LIN {X 0,Y 496.76,Z 265.856,A -85,B 0,C 180,E1 24154.304,E2 24154.304} C_VEL
LIN {X 0,Y 496.744,Z 265.83,A -85,B 0,C 180,E1 24150.745,E2 24150.745} C_VEL
LIN {X 0,Y 496.768,Z 265.857,A -85,B 0,C 180,E1 24147.316,E2 24147.316} C_VEL
LIN {X 0,Y 496.772,Z 265.855,A -85,B 0,C 180,E1 24143.686,E2 24143.686} C_VEL
LIN {X 0,Y 496.741,Z 265.856,A -85,B 0,C 180,E1 24140.256,E2 24140.256} C_VEL
LIN {X 0,Y 496.732,Z 265.859,A -85,B 0,C 180,E1 24136.645,E2 24136.645} C_VEL
LIN {X 0,Y 496.759,Z 265.856,A -85,B 0,C 180,E1 24133.147,E2 24133.147} C_VEL
LIN {X 0,Y 496.765,Z 265.845,A -85,B 0,C 180,E1 24129.617,E2 24129.617} C_VEL
LIN {X 0,Y 496.72,Z 265.85,A -85,B 0,C 180,E1 24126.24,E2 24126.24} C_VEL
LIN {X 0,Y 496.719,Z 265.855,A -85,B 0,C 180,E1 24122.654,E2 24122.654} C_VEL
LIN {X 0,Y 496.76,Z 265.86,A -85,B 0,C 180,E1 24119.193,E2 24119.193} C_VEL
LIN {X 0,Y 496.733,Z 265.855,A -85,B 0,C 180,E1 24115.729,E2 24115.729} C_VEL
LIN {X 0,Y 496.699,Z 265.854,A -85,B 0,C 180,E1 24112.365,E2 24112.365} C_VEL
LIN {X 0,Y 496.73,Z 265.851,A -85,B 0,C 180,E1 24108.976,E2 24108.976} C_VEL
LIN {X 0,Y 496.727,Z 265.86,A -85,B 0,C 180,E1 24105.546,E2 24105.546} C_VEL
LIN {X 0,Y 496.69,Z 265.861,A -85,B 0,C 180,E1 24102.183,E2 24102.183} C_VEL
LIN {X 0,Y 496.72,Z 265.86,A -85,B 0,C 180,E1 24098.742,E2 24098.742} C_VEL
LIN {X 0,Y 496.747,Z 265.859,A -85,B 0,C 180,E1 24095.377,E2 24095.377} C_VEL
LIN {X 0,Y 496.706,Z 265.861,A -85,B 0,C 180,E1 24092.029,E2 24092.029} C_VEL
LIN {X 0,Y 496.724,Z 265.83,A -85,B 0,C 180,E1 24088.578,E2 24088.578} C_VEL
LIN {X 0,Y 496.766,Z 265.852,A -85,B 0,C 180,E1 24085.137,E2 24085.137} C_VEL
LIN {X 0,Y 496.729,Z 265.852,A -85,B 0,C 180,E1 24081.686,E2 24081.686} C_VEL
LIN {X 0,Y 496.723,Z 265.835,A -85,B 0,C 180,E1 24078.138,E2 24078.138} C_VEL
LIN {X 0,Y 496.761,Z 265.831,A -85,B 0,C 180,E1 24074.724,E2 24074.724} C_VEL
LIN {X 0,Y 496.765,Z 266.073,A -85,B 0,C 180,E1 24073.733,E2 24073.733} C_VEL
LIN {X 0,Y 498.202,Z 269.541,A -85,B 0,C 180,E1 24073.238,E2 24073.238} C_VEL
LIN {X 0,Y 506.88,Z 288.7,A -85,B 0,C 180,E1 24070.845,E2 24070.845} C_VEL
LIN {X 0,Y 512.314,Z 301.504,A -85,B 0,C 180,E1 24069.366,E2 24069.366} C_VEL
LIN {X 0,Y 512.445,Z 304.432,A -85,B 0,C 180,E1 24069.211,E2 24069.211} C_VEL
LIN {X 0,Y 515.554,Z 323.753,A -85,B 0,C 180,E1 24068.621,E2 24068.621} C_VEL
LIN {X 0,Y 512.644,Z 536.307,A -85,B 0,C 180,E1 24065.312,E2 24065.312} C_VEL
LIN {X 0,Y 511.651,Z 609.629,A -85,B 0,C 180,E1 24064.168,E2 24064.168} C_VEL
LIN {X 0,Y 510.839,Z 630.079,A -85,B 0,C 180,E1 24063.658,E2 24063.658} C_VEL
LIN {X 0,Y 509.734,Z 651.77,A -85,B 0,C 180,E1 24062.909,E2 24062.909} C_VEL
LIN {X 0,Y 508.491,Z 672.18,A -85,B 0,C 180,E1 24061.999,E2 24061.999} C_VEL
LIN {X 0,Y 507.033,Z 691.752,A -85,B 0,C 180,E1 24060.91,E2 24060.91} C_VEL
LIN {X 0,Y 505.464,Z 711.909,A -85,B 0,C 180,E1 24059.555,E2 24059.555} C_VEL
LIN {X 0,Y 503.931,Z 730.052,A -85,B 0,C 180,E1 24058.113,E2 24058.113} C_VEL
LIN {X 0,Y 502.359,Z 748.13,A -85,B 0,C 180,E1 24056.409,E2 24056.409} C_VEL
LIN {X 0,Y 500.871,Z 765.167,A -85,B 0,C 180,E1 24054.532,E2 24054.532} C_VEL
LIN {X 0,Y 499.613,Z 780.33,A -85,B 0,C 180,E1 24052.596,E2 24052.596} C_VEL
LIN {X 0,Y 498.485,Z 794.868,A -85,B 0,C 180,E1 24050.426,E2 24050.426} C_VEL
LIN {X 0,Y 497.624,Z 807.187,A -85,B 0,C 180,E1 24048.266,E2 24048.266} C_VEL
LIN {X 0,Y 496.93,Z 818.784,A -85,B 0,C 180,E1 24045.881,E2 24045.881} C_VEL
LIN {X 0,Y 496.465,Z 828.431,A -85,B 0,C 180,E1 24043.51,E2 24043.51} C_VEL
LIN {X 0,Y 496.159,Z 836.434,A -85,B 0,C 180,E1 24041.069,E2 24041.069} C_VEL
LIN {X 0,Y 495.997,Z 842.892,A -85,B 0,C 180,E1 24038.579,E2 24038.579} C_VEL
LIN {X 0,Y 495.935,Z 847.43,A -85,B 0,C 180,E1 24036.25,E2 24036.25} C_VEL
LIN {X 0,Y 495.907,Z 850.56,A -85,B 0,C 180,E1 24033.815,E2 24033.815} C_VEL
LIN {X 0,Y 495.902,Z 852.237,A -85,B 0,C 180,E1 24031.386,E2 24031.386} C_VEL
LIN {X 0,Y 495.909,Z 852.327,A -85,B 0,C 180,E1 24029.076,E2 24029.076} C_VEL
LIN {X 0,Y 495.911,Z 850.898,A -85,B 0,C 180,E1 24026.532,E2 24026.532} C_VEL
LIN {X 0,Y 495.931,Z 847.98,A -85,B 0,C 180,E1 24024.098,E2 24024.098} C_VEL
LIN {X 0,Y 496,Z 843.399,A -85,B 0,C 180,E1 24021.655,E2 24021.655} C_VEL
LIN {X 0,Y 496.141,Z 837.235,A -85,B 0,C 180,E1 24019.198,E2 24019.198} C_VEL
LIN {X 0,Y 496.403,Z 829.665,A -85,B 0,C 180,E1 24016.844,E2 24016.844} C_VEL
LIN {X 0,Y 496.836,Z 820.328,A -85,B 0,C 180,E1 24014.476,E2 24014.476} C_VEL
LIN {X 0,Y 497.459,Z 809.727,A -85,B 0,C 180,E1 24012.212,E2 24012.212} C_VEL
LIN {X 0,Y 498.274,Z 797.763,A -85,B 0,C 180,E1 24010.055,E2 24010.055} C_VEL
LIN {X 0,Y 499.339,Z 783.717,A -85,B 0,C 180,E1 24007.887,E2 24007.887} C_VEL
LIN {X 0,Y 500.624,Z 768.208,A -85,B 0,C 180,E1 24005.832,E2 24005.832} C_VEL
LIN {X 0,Y 501.995,Z 752.25,A -85,B 0,C 180,E1 24004.012,E2 24004.012} C_VEL
LIN {X 0,Y 503.516,Z 734.772,A -85,B 0,C 180,E1 24002.312,E2 24002.312} C_VEL
LIN {X 0,Y 505.136,Z 715.755,A -85,B 0,C 180,E1 24000.732,E2 24000.732} C_VEL
LIN {X 0,Y 506.688,Z 696.76,A -85,B 0,C 180,E1 23999.396,E2 23999.396} C_VEL
LIN {X 0,Y 508.188,Z 676.137,A -85,B 0,C 180,E1 23998.207,E2 23998.207} C_VEL
LIN {X 0,Y 509.534,Z 655.455,A -85,B 0,C 180,E1 23997.242,E2 23997.242} C_VEL
LIN {X 0,Y 510.643,Z 634.593,A -85,B 0,C 180,E1 23996.473,E2 23996.473} C_VEL
LIN {X 0,Y 511.474,Z 614.158,A -85,B 0,C 180,E1 23995.932,E2 23995.932} C_VEL
LIN {X 0,Y 512.059,Z 584.884,A -85,B 0,C 180,E1 23995.426,E2 23995.426} C_VEL
LIN {X 0,Y 514.855,Z 371.498,A -85,B 0,C 180,E1 23992.134,E2 23992.134} C_VEL
LIN {X 0,Y 515.386,Z 321.569,A -85,B 0,C 180,E1 23991.328,E2 23991.328} C_VEL
LIN {X 0,Y 512.272,Z 302.49,A -85,B 0,C 180,E1 23990.703,E2 23990.703} C_VEL
LIN {X 0,Y 512.096,Z 300.679,A -85,B 0,C 180,E1 23990.552,E2 23990.552} C_VEL
LIN {X 0,Y 502.008,Z 277.659,A -85,B 0,C 180,E1 23987.809,E2 23987.809} C_VEL
LIN {X 0,Y 496.796,Z 266.243,A -85,B 0,C 180,E1 23986.311,E2 23986.311} C_VEL
LIN {X 0,Y 496.743,Z 265.832,A -85,B 0,C 180,E1 23985.537,E2 23985.537} C_VEL
LIN {X 0,Y 496.723,Z 265.836,A -85,B 0,C 180,E1 23982.034,E2 23982.034} C_VEL
LIN {X 0,Y 496.753,Z 265.852,A -85,B 0,C 180,E1 23978.606,E2 23978.606} C_VEL
LIN {X 0,Y 496.758,Z 265.848,A -85,B 0,C 180,E1 23975.145,E2 23975.145} C_VEL
LIN {X 0,Y 496.712,Z 265.833,A -85,B 0,C 180,E1 23971.694,E2 23971.694} C_VEL
LIN {X 0,Y 496.713,Z 265.861,A -85,B 0,C 180,E1 23968.101,E2 23968.101} C_VEL
LIN {X 0,Y 496.76,Z 265.86,A -85,B 0,C 180,E1 23964.749,E2 23964.749} C_VEL
LIN {X 0,Y 496.712,Z 265.86,A -85,B 0,C 180,E1 23961.367,E2 23961.367} C_VEL
LIN {X 0,Y 496.695,Z 265.861,A -85,B 0,C 180,E1 23957.938,E2 23957.938} C_VEL
LIN {X 0,Y 496.733,Z 265.858,A -85,B 0,C 180,E1 23954.496,E2 23954.496} C_VEL
LIN {X 0,Y 496.725,Z 265.851,A -85,B 0,C 180,E1 23951.024,E2 23951.024} C_VEL
LIN {X 0,Y 496.695,Z 265.855,A -85,B 0,C 180,E1 23947.635,E2 23947.635} C_VEL
LIN {X 0,Y 496.721,Z 265.856,A -85,B 0,C 180,E1 23944.155,E2 23944.155} C_VEL
LIN {X 0,Y 496.767,Z 265.859,A -85,B 0,C 180,E1 23940.692,E2 23940.692} C_VEL
LIN {X 0,Y 496.72,Z 265.855,A -85,B 0,C 180,E1 23937.231,E2 23937.231} C_VEL
LIN {X 0,Y 496.717,Z 265.85,A -85,B 0,C 180,E1 23933.759,E2 23933.759} C_VEL
LIN {X 0,Y 496.764,Z 265.846,A -85,B 0,C 180,E1 23930.383,E2 23930.383} C_VEL
LIN {X 0,Y 496.753,Z 265.858,A -85,B 0,C 180,E1 23926.853,E2 23926.853} C_VEL
LIN {X 0,Y 496.728,Z 265.858,A -85,B 0,C 180,E1 23923.391,E2 23923.391} C_VEL
LIN {X 0,Y 496.745,Z 265.855,A -85,B 0,C 180,E1 23919.867,E2 23919.867} C_VEL
LIN {X 0,Y 496.771,Z 265.856,A -85,B 0,C 180,E1 23916.388,E2 23916.388} C_VEL
LIN {X 0,Y 496.761,Z 265.853,A -85,B 0,C 180,E1 23912.813,E2 23912.813} C_VEL
LIN {X 0,Y 496.74,Z 265.832,A -85,B 0,C 180,E1 23909.386,E2 23909.386} C_VEL
LIN {X 0,Y 496.762,Z 265.855,A -85,B 0,C 180,E1 23905.814,E2 23905.814} C_VEL
LIN {X 0,Y 496.762,Z 265.83,A -85,B 0,C 180,E1 23902.274,E2 23902.274} C_VEL
LIN {X 0,Y 496.768,Z 265.836,A -85,B 0,C 180,E1 23898.687,E2 23898.687} C_VEL
LIN {X 0,Y 496.758,Z 265.857,A -85,B 0,C 180,E1 23895.05,E2 23895.05} C_VEL
LIN {X 0,Y 496.765,Z 265.859,A -85,B 0,C 180,E1 23891.466,E2 23891.466} C_VEL
LIN {X 0,Y 496.819,Z 266.17,A -85,B 0,C 180,E1 23890.648,E2 23890.648} C_VEL
LIN {X 0,Y 505.817,Z 287.439,A -85,B 0,C 180,E1 23887.75,E2 23887.75} C_VEL
LIN {X 0,Y 507.172,Z 290.873,A -85,B 0,C 180,E1 23887.316,E2 23887.316} C_VEL
LIN {X 0,Y 507.772,Z 294.918,A -85,B 0,C 180,E1 23886.901,E2 23886.901} C_VEL
LIN {X 0,Y 506.892,Z 301.33,A -85,B 0,C 180,E1 23886.41,E2 23886.41} C_VEL
LIN {X 0,Y 502.273,Z 317.887,A -85,B 0,C 180,E1 23885.352,E2 23885.352} C_VEL
LIN {X 0,Y 501.917,Z 320.739,A -85,B 0,C 180,E1 23885.132,E2 23885.132} C_VEL
LIN {X 0,Y 501.604,Z 327.881,A -85,B 0,C 180,E1 23884.576,E2 23884.576} C_VEL
LIN {X 0,Y 505.479,Z 350.471,A -85,B 0,C 180,E1 23883.865,E2 23883.865} C_VEL
LIN {X 0,Y 502.237,Z 583.059,A -85,B 0,C 180,E1 23880.294,E2 23880.294} C_VEL
LIN {X 0,Y 501.63,Z 603.88,A -85,B 0,C 180,E1 23879.854,E2 23879.854} C_VEL
LIN {X 0,Y 500.665,Z 623.703,A -85,B 0,C 180,E1 23879.22,E2 23879.22} C_VEL
LIN {X 0,Y 499.463,Z 643.041,A -85,B 0,C 180,E1 23878.387,E2 23878.387} C_VEL
LIN {X 0,Y 498.088,Z 661.685,A -85,B 0,C 180,E1 23877.366,E2 23877.366} C_VEL
LIN {X 0,Y 496.606,Z 679.561,A -85,B 0,C 180,E1 23876.163,E2 23876.163} C_VEL
LIN {X 0,Y 495.015,Z 697.298,A -85,B 0,C 180,E1 23874.715,E2 23874.715} C_VEL
LIN {X 0,Y 493.413,Z 714.532,A -85,B 0,C 180,E1 23873.022,E2 23873.022} C_VEL
LIN {X 0,Y 491.984,Z 730.027,A -85,B 0,C 180,E1 23871.207,E2 23871.207} C_VEL
LIN {X 0,Y 490.748,Z 744.004,A -85,B 0,C 180,E1 23869.272,E2 23869.272} C_VEL
LIN {X 0,Y 489.675,Z 758.025,A -85,B 0,C 180,E1 23866.977,E2 23866.977} C_VEL
LIN {X 0,Y 488.978,Z 769.274,A -85,B 0,C 180,E1 23864.809,E2 23864.809} C_VEL
LIN {X 0,Y 488.472,Z 779.247,A -85,B 0,C 180,E1 23862.478,E2 23862.478} C_VEL
LIN {X 0,Y 488.166,Z 787.28,A -85,B 0,C 180,E1 23860.145,E2 23860.145} C_VEL
LIN {X 0,Y 488.015,Z 793.376,A -85,B 0,C 180,E1 23857.89,E2 23857.89} C_VEL
LIN {X 0,Y 487.931,Z 798.008,A -85,B 0,C 180,E1 23855.527,E2 23855.527} C_VEL
LIN {X 0,Y 487.909,Z 800.962,A -85,B 0,C 180,E1 23853.172,E2 23853.172} C_VEL
LIN {X 0,Y 487.907,Z 802.359,A -85,B 0,C 180,E1 23850.704,E2 23850.704} C_VEL
LIN {X 0,Y 487.902,Z 802.102,A -85,B 0,C 180,E1 23848.356,E2 23848.356} C_VEL
LIN {X 0,Y 487.918,Z 800.255,A -85,B 0,C 180,E1 23846.005,E2 23846.005} C_VEL
LIN {X 0,Y 487.953,Z 796.675,A -85,B 0,C 180,E1 23843.622,E2 23843.622} C_VEL
LIN {X 0,Y 488.053,Z 791.516,A -85,B 0,C 180,E1 23841.281,E2 23841.281} C_VEL
LIN {X 0,Y 488.258,Z 784.528,A -85,B 0,C 180,E1 23838.902,E2 23838.902} C_VEL
LIN {X 0,Y 488.621,Z 776.086,A -85,B 0,C 180,E1 23836.631,E2 23836.631} C_VEL
LIN {X 0,Y 489.198,Z 765.655,A -85,B 0,C 180,E1 23834.349,E2 23834.349} C_VEL
LIN {X 0,Y 490.041,Z 752.956,A -85,B 0,C 180,E1 23832.056,E2 23832.056} C_VEL
LIN {X 0,Y 491.123,Z 739.689,A -85,B 0,C 180,E1 23830,E2 23830} C_VEL
LIN {X 0,Y 492.441,Z 724.859,A -85,B 0,C 180,E1 23828.063,E2 23828.063} C_VEL
LIN {X 0,Y 493.859,Z 709.496,A -85,B 0,C 180,E1 23826.368,E2 23826.368} C_VEL
LIN {X 0,Y 495.425,Z 692.653,A -85,B 0,C 180,E1 23824.797,E2 23824.797} C_VEL
LIN {X 0,Y 497,Z 674.858,A -85,B 0,C 180,E1 23823.41,E2 23823.41} C_VEL
LIN {X 0,Y 498.465,Z 657.122,A -85,B 0,C 180,E1 23822.267,E2 23822.267} C_VEL
LIN {X 0,Y 499.773,Z 638.535,A -85,B 0,C 180,E1 23821.306,E2 23821.306} C_VEL
LIN {X 0,Y 500.896,Z 619.188,A -85,B 0,C 180,E1 23820.53,E2 23820.53} C_VEL
LIN {X 0,Y 501.8,Z 598.35,A -85,B 0,C 180,E1 23819.922,E2 23819.922} C_VEL
LIN {X 0,Y 502.38,Z 574.514,A -85,B 0,C 180,E1 23819.48,E2 23819.48} C_VEL
LIN {X 0,Y 505.455,Z 349.374,A -85,B 0,C 180,E1 23816.024,E2 23816.024} C_VEL
LIN {X 0,Y 501.532,Z 326.8,A -85,B 0,C 180,E1 23815.274,E2 23815.274} C_VEL
LIN {X 0,Y 503.113,Z 301.394,A -85,B 0,C 180,E1 23813.169,E2 23813.169} C_VEL
LIN {X 0,Y 495.083,Z 281.538,A -85,B 0,C 180,E1 23810.578,E2 23810.578} C_VEL
LIN {X 0,Y 488.87,Z 267.138,A -85,B 0,C 180,E1 23808.498,E2 23808.498} C_VEL
LIN {X 0,Y 488.825,Z 266.818,A -85,B 0,C 180,E1 23806.426,E2 23806.426} C_VEL
LIN {X 0,Y 488.818,Z 266.819,A -85,B 0,C 180,E1 23802.924,E2 23802.924} C_VEL
LIN {X 0,Y 488.831,Z 266.843,A -85,B 0,C 180,E1 23799.352,E2 23799.352} C_VEL
LIN {X 0,Y 488.824,Z 266.832,A -85,B 0,C 180,E1 23795.659,E2 23795.659} C_VEL
LIN {X 0,Y 488.823,Z 266.82,A -85,B 0,C 180,E1 23792.128,E2 23792.128} C_VEL
LIN {X 0,Y 488.807,Z 266.847,A -85,B 0,C 180,E1 23788.597,E2 23788.597} C_VEL
LIN {X 0,Y 488.817,Z 266.846,A -85,B 0,C 180,E1 23785.026,E2 23785.026} C_VEL
LIN {X 0,Y 488.832,Z 266.838,A -85,B 0,C 180,E1 23781.467,E2 23781.467} C_VEL
LIN {X 0,Y 488.822,Z 266.836,A -85,B 0,C 180,E1 23777.868,E2 23777.868} C_VEL
LIN {X 0,Y 488.792,Z 266.837,A -85,B 0,C 180,E1 23774.331,E2 23774.331} C_VEL
LIN {X 0,Y 488.79,Z 266.836,A -85,B 0,C 180,E1 23770.728,E2 23770.728} C_VEL
LIN {X 0,Y 488.828,Z 266.842,A -85,B 0,C 180,E1 23767.252,E2 23767.252} C_VEL
LIN {X 0,Y 488.807,Z 266.846,A -85,B 0,C 180,E1 23763.753,E2 23763.753} C_VEL
LIN {X 0,Y 488.771,Z 266.847,A -85,B 0,C 180,E1 23760.352,E2 23760.352} C_VEL
LIN {X 0,Y 488.785,Z 266.842,A -85,B 0,C 180,E1 23756.834,E2 23756.834} C_VEL
LIN {X 0,Y 488.827,Z 266.838,A -85,B 0,C 180,E1 23753.305,E2 23753.305} C_VEL
LIN {X 0,Y 488.77,Z 266.85,A -85,B 0,C 180,E1 23749.868,E2 23749.868} C_VEL
LIN {X 0,Y 488.752,Z 266.85,A -85,B 0,C 180,E1 23746.336,E2 23746.336} C_VEL
LIN {X 0,Y 488.794,Z 266.85,A -85,B 0,C 180,E1 23742.992,E2 23742.992} C_VEL
LIN {X 0,Y 488.79,Z 266.844,A -85,B 0,C 180,E1 23739.526,E2 23739.526} C_VEL
LIN {X 0,Y 488.762,Z 266.847,A -85,B 0,C 180,E1 23736.106,E2 23736.106} C_VEL
LIN {X 0,Y 488.783,Z 266.849,A -85,B 0,C 180,E1 23732.594,E2 23732.594} C_VEL
LIN {X 0,Y 488.831,Z 266.813,A -85,B 0,C 180,E1 23729.11,E2 23729.11} C_VEL
LIN {X 0,Y 488.801,Z 266.851,A -85,B 0,C 180,E1 23725.52,E2 23725.52} C_VEL
LIN {X 0,Y 488.779,Z 266.834,A -85,B 0,C 180,E1 23721.995,E2 23721.995} C_VEL
LIN {X 0,Y 488.799,Z 266.819,A -85,B 0,C 180,E1 23718.473,E2 23718.473} C_VEL
LIN {X 0,Y 488.829,Z 266.819,A -85,B 0,C 180,E1 23714.951,E2 23714.951} C_VEL
LIN {X 0,Y 488.877,Z 267.302,A -85,B 0,C 180,E1 23714.435,E2 23714.435} C_VEL
LIN {X 0,Y 497.975,Z 287.252,A -85,B 0,C 180,E1 23711.804,E2 23711.804} C_VEL
LIN {X 0,Y 505.312,Z 303.93,A -85,B 0,C 180,E1 23709.827,E2 23709.827} C_VEL
LIN {X 0,Y 506.077,Z 306.304,A -85,B 0,C 180,E1 23709.716,E2 23709.716} C_VEL
LIN {X 0,Y 509.065,Z 325.262,A -85,B 0,C 180,E1 23709.128,E2 23709.128} C_VEL
LIN {X 0,Y 505.837,Z 535.278,A -85,B 0,C 180,E1 23705.801,E2 23705.801} C_VEL
LIN {X 0,Y 504.715,Z 609.546,A -85,B 0,C 180,E1 23704.623,E2 23704.623} C_VEL
LIN {X 0,Y 503.838,Z 631.178,A -85,B 0,C 180,E1 23704.08,E2 23704.08} C_VEL
LIN {X 0,Y 502.733,Z 652.958,A -85,B 0,C 180,E1 23703.327,E2 23703.327} C_VEL
LIN {X 0,Y 501.529,Z 673.25,A -85,B 0,C 180,E1 23702.43,E2 23702.43} C_VEL
LIN {X 0,Y 500.052,Z 691.983,A -85,B 0,C 180,E1 23701.374,E2 23701.374} C_VEL
LIN {X 0,Y 498.309,Z 712.502,A -85,B 0,C 180,E1 23699.974,E2 23699.974} C_VEL
LIN {X 0,Y 496.645,Z 730.759,A -85,B 0,C 180,E1 23698.498,E2 23698.498} C_VEL
LIN {X 0,Y 494.933,Z 748.869,A -85,B 0,C 180,E1 23696.758,E2 23696.758} C_VEL
LIN {X 0,Y 493.328,Z 765.673,A -85,B 0,C 180,E1 23694.869,E2 23694.869} C_VEL
LIN {X 0,Y 491.921,Z 781.18,A -85,B 0,C 180,E1 23692.843,E2 23692.843} C_VEL
LIN {X 0,Y 490.705,Z 795.633,A -85,B 0,C 180,E1 23690.64,E2 23690.64} C_VEL
LIN {X 0,Y 489.724,Z 808.455,A -85,B 0,C 180,E1 23688.325,E2 23688.325} C_VEL
LIN {X 0,Y 488.981,Z 819.813,A -85,B 0,C 180,E1 23685.902,E2 23685.902} C_VEL
LIN {X 0,Y 488.486,Z 829.26,A -85,B 0,C 180,E1 23683.493,E2 23683.493} C_VEL
LIN {X 0,Y 488.176,Z 836.882,A -85,B 0,C 180,E1 23681.1,E2 23681.1} C_VEL
LIN {X 0,Y 488.003,Z 843.146,A -85,B 0,C 180,E1 23678.602,E2 23678.602} C_VEL
LIN {X 0,Y 487.937,Z 847.823,A -85,B 0,C 180,E1 23676.117,E2 23676.117} C_VEL
LIN {X 0,Y 487.908,Z 850.799,A -85,B 0,C 180,E1 23673.63,E2 23673.63} C_VEL
LIN {X 0,Y 487.911,Z 852.304,A -85,B 0,C 180,E1 23671.057,E2 23671.057} C_VEL
LIN {X 0,Y 487.905,Z 852.258,A -85,B 0,C 180,E1 23668.708,E2 23668.708} C_VEL
LIN {X 0,Y 487.907,Z 850.671,A -85,B 0,C 180,E1 23666.24,E2 23666.24} C_VEL
LIN {X 0,Y 487.937,Z 847.633,A -85,B 0,C 180,E1 23663.765,E2 23663.765} C_VEL
LIN {X 0,Y 488.003,Z 843.145,A -85,B 0,C 180,E1 23661.398,E2 23661.398} C_VEL
LIN {X 0,Y 488.184,Z 836.663,A -85,B 0,C 180,E1 23658.826,E2 23658.826} C_VEL
LIN {X 0,Y 488.51,Z 828.85,A -85,B 0,C 180,E1 23656.387,E2 23656.387} C_VEL
LIN {X 0,Y 489.028,Z 819.118,A -85,B 0,C 180,E1 23653.935,E2 23653.935} C_VEL
LIN {X 0,Y 489.77,Z 807.821,A -85,B 0,C 180,E1 23651.553,E2 23651.553} C_VEL
LIN {X 0,Y 490.704,Z 795.633,A -85,B 0,C 180,E1 23649.36,E2 23649.36} C_VEL
LIN {X 0,Y 491.921,Z 781.18,A -85,B 0,C 180,E1 23647.157,E2 23647.157} C_VEL
LIN {X 0,Y 493.328,Z 765.674,A -85,B 0,C 180,E1 23645.131,E2 23645.131} C_VEL
LIN {X 0,Y 494.947,Z 748.704,A -85,B 0,C 180,E1 23643.226,E2 23643.226} C_VEL
LIN {X 0,Y 496.644,Z 730.761,A -85,B 0,C 180,E1 23641.502,E2 23641.502} C_VEL
LIN {X 0,Y 498.311,Z 712.507,A -85,B 0,C 180,E1 23640.026,E2 23640.026} C_VEL
LIN {X 0,Y 500.053,Z 691.986,A -85,B 0,C 180,E1 23638.626,E2 23638.626} C_VEL
LIN {X 0,Y 501.529,Z 673.25,A -85,B 0,C 180,E1 23637.57,E2 23637.57} C_VEL
LIN {X 0,Y 502.778,Z 652.163,A -85,B 0,C 180,E1 23636.64,E2 23636.64} C_VEL
LIN {X 0,Y 503.902,Z 629.839,A -85,B 0,C 180,E1 23635.882,E2 23635.882} C_VEL
LIN {X 0,Y 504.741,Z 608.427,A -85,B 0,C 180,E1 23635.356,E2 23635.356} C_VEL
LIN {X 0,Y 508.171,Z 379.59,A -85,B 0,C 180,E1 23631.748,E2 23631.748} C_VEL
LIN {X 0,Y 508.918,Z 323.091,A -85,B 0,C 180,E1 23630.822,E2 23630.822} C_VEL
LIN {X 0,Y 505.558,Z 304.395,A -85,B 0,C 180,E1 23630.205,E2 23630.205} C_VEL
LIN {X 0,Y 503.403,Z 299.648,A -85,B 0,C 180,E1 23629.702,E2 23629.702} C_VEL
LIN {X 0,Y 494.096,Z 278.623,A -85,B 0,C 180,E1 23627.1,E2 23627.1} C_VEL
LIN {X 0,Y 488.868,Z 267.247,A -85,B 0,C 180,E1 23625.556,E2 23625.556} C_VEL
LIN {X 0,Y 488.828,Z 266.821,A -85,B 0,C 180,E1 23624.883,E2 23624.883} C_VEL
LIN {X 0,Y 488.811,Z 266.818,A -85,B 0,C 180,E1 23621.351,E2 23621.351} C_VEL
LIN {X 0,Y 488.781,Z 266.834,A -85,B 0,C 180,E1 23618.005,E2 23618.005} C_VEL
LIN {X 0,Y 488.802,Z 266.851,A -85,B 0,C 180,E1 23614.48,E2 23614.48} C_VEL
LIN {X 0,Y 488.831,Z 266.812,A -85,B 0,C 180,E1 23610.89,E2 23610.89} C_VEL
LIN {X 0,Y 488.783,Z 266.849,A -85,B 0,C 180,E1 23607.404,E2 23607.404} C_VEL
LIN {X 0,Y 488.763,Z 266.846,A -85,B 0,C 180,E1 23603.88,E2 23603.88} C_VEL
LIN {X 0,Y 488.793,Z 266.843,A -85,B 0,C 180,E1 23600.472,E2 23600.472} C_VEL
LIN {X 0,Y 488.796,Z 266.85,A -85,B 0,C 180,E1 23597.008,E2 23597.008} C_VEL
LIN {X 0,Y 488.752,Z 266.85,A -85,B 0,C 180,E1 23593.607,E2 23593.607} C_VEL
LIN {X 0,Y 488.762,Z 266.85,A -85,B 0,C 180,E1 23590.013,E2 23590.013} C_VEL
LIN {X 0,Y 488.818,Z 266.84,A -85,B 0,C 180,E1 23586.577,E2 23586.577} C_VEL
LIN {X 0,Y 488.789,Z 266.841,A -85,B 0,C 180,E1 23583.048,E2 23583.048} C_VEL
LIN {X 0,Y 488.768,Z 266.847,A -85,B 0,C 180,E1 23579.648,E2 23579.648} C_VEL
LIN {X 0,Y 488.796,Z 266.846,A -85,B 0,C 180,E1 23576.129,E2 23576.129} C_VEL
LIN {X 0,Y 488.838,Z 266.843,A -85,B 0,C 180,E1 23572.596,E2 23572.596} C_VEL
LIN {X 0,Y 488.798,Z 266.838,A -85,B 0,C 180,E1 23569.033,E2 23569.033} C_VEL
LIN {X 0,Y 488.786,Z 266.838,A -85,B 0,C 180,E1 23565.548,E2 23565.548} C_VEL
LIN {X 0,Y 488.821,Z 266.836,A -85,B 0,C 180,E1 23562.132,E2 23562.132} C_VEL
LIN {X 0,Y 488.834,Z 266.839,A -85,B 0,C 180,E1 23558.523,E2 23558.523} C_VEL
LIN {X 0,Y 488.813,Z 266.847,A -85,B 0,C 180,E1 23554.949,E2 23554.949} C_VEL
LIN {X 0,Y 488.802,Z 266.847,A -85,B 0,C 180,E1 23551.343,E2 23551.343} C_VEL
LIN {X 0,Y 488.822,Z 266.818,A -85,B 0,C 180,E1 23547.864,E2 23547.864} C_VEL
LIN {X 0,Y 488.827,Z 266.832,A -85,B 0,C 180,E1 23544.293,E2 23544.293} C_VEL
LIN {X 0,Y 488.832,Z 266.842,A -85,B 0,C 180,E1 23540.637,E2 23540.637} C_VEL
LIN {X 0,Y 488.814,Z 266.819,A -85,B 0,C 180,E1 23537.067,E2 23537.067} C_VEL
LIN {X 0,Y 488.819,Z 266.819,A -85,B 0,C 180,E1 23533.436,E2 23533.436} C_VEL
LIN {X 0,Y 488.865,Z 267.126,A -85,B 0,C 180,E1 23531.412,E2 23531.412} C_VEL
LIN {X 0,Y 491.5,Z 273.545,A -85,B 0,C 180,E1 23530.46,E2 23530.46} C_VEL
LIN {X 0,Y 498.623,Z 290.133,A -85,B 0,C 180,E1 23528.181,E2 23528.181} C_VEL
LIN {X 0,Y 503.166,Z 301.796,A -85,B 0,C 180,E1 23526.699,E2 23526.699} C_VEL
LIN {X 0,Y 501.917,Z 320.739,A -85,B 0,C 180,E1 23525.132,E2 23525.132} C_VEL
LIN {X 0,Y 501.615,Z 326.574,A -85,B 0,C 180,E1 23524.772,E2 23524.772} C_VEL
LIN {X 0,Y 501.194,Z 334.058,A -85,B 0,C 180,E1 23524.531,E2 23524.531} C_VEL
LIN {X 0,Y 500.135,Z 343.047,A -85,B 0,C 180,E1 23524.446,E2 23524.446} C_VEL
LIN {X 0,Y 499.043,Z 353.304,A -85,B 0,C 180,E1 23524.367,E2 23524.367} C_VEL
LIN {X 0,Y 498.975,Z 355.582,A -85,B 0,C 180,E1 23524.334,E2 23524.334} C_VEL
LIN {X 0,Y 495.627,Z 585.263,A -85,B 0,C 180,E1 23520.786,E2 23520.786} C_VEL
LIN {X 0,Y 494.992,Z 605.301,A -85,B 0,C 180,E1 23520.346,E2 23520.346} C_VEL
LIN {X 0,Y 493.977,Z 624.896,A -85,B 0,C 180,E1 23519.708,E2 23519.708} C_VEL
LIN {X 0,Y 492.704,Z 643.755,A -85,B 0,C 180,E1 23518.879,E2 23518.879} C_VEL
LIN {X 0,Y 491.221,Z 662.302,A -85,B 0,C 180,E1 23517.848,E2 23517.848} C_VEL
LIN {X 0,Y 489.616,Z 680.13,A -85,B 0,C 180,E1 23516.63,E2 23516.63} C_VEL
LIN {X 0,Y 487.897,Z 697.838,A -85,B 0,C 180,E1 23515.165,E2 23515.165} C_VEL
LIN {X 0,Y 486.157,Z 714.834,A -85,B 0,C 180,E1 23513.469,E2 23513.469} C_VEL
LIN {X 0,Y 484.598,Z 729.944,A -85,B 0,C 180,E1 23511.673,E2 23511.673} C_VEL
LIN {X 0,Y 483.216,Z 744.054,A -85,B 0,C 180,E1 23509.699,E2 23509.699} C_VEL
LIN {X 0,Y 482.103,Z 756.593,A -85,B 0,C 180,E1 23507.625,E2 23507.625} C_VEL
LIN {X 0,Y 481.225,Z 767.881,A -85,B 0,C 180,E1 23505.405,E2 23505.405} C_VEL
LIN {X 0,Y 480.597,Z 778.13,A -85,B 0,C 180,E1 23502.984,E2 23502.984} C_VEL
LIN {X 0,Y 480.243,Z 786.238,A -85,B 0,C 180,E1 23500.673,E2 23500.673} C_VEL
LIN {X 0,Y 480.042,Z 792.805,A -85,B 0,C 180,E1 23498.263,E2 23498.263} C_VEL
LIN {X 0,Y 479.947,Z 797.596,A -85,B 0,C 180,E1 23495.859,E2 23495.859} C_VEL
LIN {X 0,Y 479.908,Z 800.734,A -85,B 0,C 180,E1 23493.464,E2 23493.464} C_VEL
LIN {X 0,Y 479.91,Z 802.291,A -85,B 0,C 180,E1 23491.074,E2 23491.074} C_VEL
LIN {X 0,Y 479.905,Z 802.265,A -85,B 0,C 180,E1 23488.687,E2 23488.687} C_VEL
LIN {X 0,Y 479.911,Z 800.594,A -85,B 0,C 180,E1 23486.297,E2 23486.297} C_VEL
LIN {X 0,Y 479.951,Z 797.337,A -85,B 0,C 180,E1 23483.901,E2 23483.901} C_VEL
LIN {X 0,Y 480.049,Z 792.424,A -85,B 0,C 180,E1 23481.496,E2 23481.496} C_VEL
LIN {X 0,Y 480.26,Z 785.742,A -85,B 0,C 180,E1 23479.079,E2 23479.079} C_VEL
LIN {X 0,Y 480.649,Z 777.089,A -85,B 0,C 180,E1 23476.65,E2 23476.65} C_VEL
LIN {X 0,Y 481.372,Z 765.964,A -85,B 0,C 180,E1 23474.087,E2 23474.087} C_VEL
LIN {X 0,Y 482.372,Z 753.684,A -85,B 0,C 180,E1 23471.761,E2 23471.761} C_VEL
LIN {X 0,Y 483.567,Z 740.482,A -85,B 0,C 180,E1 23469.674,E2 23469.674} C_VEL
LIN {X 0,Y 485.016,Z 725.757,A -85,B 0,C 180,E1 23467.709,E2 23467.709} C_VEL
LIN {X 0,Y 486.568,Z 710.563,A -85,B 0,C 180,E1 23465.992,E2 23465.992} C_VEL
LIN {X 0,Y 488.339,Z 693.186,A -85,B 0,C 180,E1 23464.34,E2 23464.34} C_VEL
LIN {X 0,Y 490.054,Z 675.422,A -85,B 0,C 180,E1 23462.937,E2 23462.937} C_VEL
LIN {X 0,Y 491.629,Z 657.752,A -85,B 0,C 180,E1 23461.781,E2 23461.781} C_VEL
LIN {X 0,Y 493.041,Z 639.23,A -85,B 0,C 180,E1 23460.81,E2 23460.81} C_VEL
LIN {X 0,Y 494.25,Z 619.896,A -85,B 0,C 180,E1 23460.022,E2 23460.022} C_VEL
LIN {X 0,Y 495.225,Z 598.831,A -85,B 0,C 180,E1 23459.401,E2 23459.401} C_VEL
LIN {X 0,Y 495.837,Z 574.579,A -85,B 0,C 180,E1 23458.949,E2 23458.949} C_VEL
LIN {X 0,Y 498.991,Z 350.623,A -85,B 0,C 180,E1 23455.492,E2 23455.492} C_VEL
LIN {X 0,Y 494.811,Z 326.867,A -85,B 0,C 180,E1 23454.697,E2 23454.697} C_VEL
LIN {X 0,Y 496.222,Z 304.676,A -85,B 0,C 180,E1 23452.836,E2 23452.836} C_VEL
LIN {X 0,Y 488.545,Z 285.708,A -85,B 0,C 180,E1 23450.311,E2 23450.311} C_VEL
LIN {X 0,Y 481.926,Z 270.887,A -85,B 0,C 180,E1 23448.144,E2 23448.144} C_VEL
LIN {X 0,Y 480.905,Z 268.038,A -85,B 0,C 180,E1 23447.685,E2 23447.685} C_VEL
LIN {X 0,Y 480.891,Z 267.836,A -85,B 0,C 180,E1 23444.315,E2 23444.315} C_VEL
LIN {X 0,Y 480.879,Z 267.826,A -85,B 0,C 180,E1 23440.633,E2 23440.633} C_VEL
LIN {X 0,Y 480.879,Z 267.803,A -85,B 0,C 180,E1 23437.022,E2 23437.022} C_VEL
LIN {X 0,Y 480.889,Z 267.828,A -85,B 0,C 180,E1 23433.435,E2 23433.435} C_VEL
LIN {X 0,Y 480.89,Z 267.814,A -85,B 0,C 180,E1 23429.797,E2 23429.797} C_VEL
LIN {X 0,Y 480.872,Z 267.825,A -85,B 0,C 180,E1 23426.288,E2 23426.288} C_VEL
LIN {X 0,Y 480.861,Z 267.826,A -85,B 0,C 180,E1 23422.624,E2 23422.624} C_VEL
LIN {X 0,Y 480.875,Z 267.826,A -85,B 0,C 180,E1 23419.053,E2 23419.053} C_VEL
LIN {X 0,Y 480.897,Z 267.829,A -85,B 0,C 180,E1 23415.434,E2 23415.434} C_VEL
LIN {X 0,Y 480.873,Z 267.834,A -85,B 0,C 180,E1 23411.879,E2 23411.879} C_VEL
LIN {X 0,Y 480.845,Z 267.836,A -85,B 0,C 180,E1 23408.37,E2 23408.37} C_VEL
LIN {X 0,Y 480.849,Z 267.838,A -85,B 0,C 180,E1 23404.771,E2 23404.771} C_VEL
LIN {X 0,Y 480.889,Z 267.824,A -85,B 0,C 180,E1 23401.311,E2 23401.311} C_VEL
LIN {X 0,Y 480.849,Z 267.834,A -85,B 0,C 180,E1 23397.855,E2 23397.855} C_VEL
LIN {X 0,Y 480.826,Z 267.838,A -85,B 0,C 180,E1 23394.391,E2 23394.391} C_VEL
LIN {X 0,Y 480.848,Z 267.84,A -85,B 0,C 180,E1 23390.908,E2 23390.908} C_VEL
LIN {X 0,Y 480.867,Z 267.83,A -85,B 0,C 180,E1 23387.39,E2 23387.39} C_VEL
LIN {X 0,Y 480.815,Z 267.83,A -85,B 0,C 180,E1 23383.944,E2 23383.944} C_VEL
LIN {X 0,Y 480.818,Z 267.832,A -85,B 0,C 180,E1 23380.313,E2 23380.313} C_VEL
LIN {X 0,Y 480.855,Z 267.829,A -85,B 0,C 180,E1 23376.859,E2 23376.859} C_VEL
LIN {X 0,Y 480.874,Z 267.829,A -85,B 0,C 180,E1 23373.313,E2 23373.313} C_VEL
LIN {X 0,Y 480.833,Z 267.818,A -85,B 0,C 180,E1 23369.885,E2 23369.885} C_VEL
LIN {X 0,Y 480.839,Z 267.84,A -85,B 0,C 180,E1 23366.276,E2 23366.276} C_VEL
LIN {X 0,Y 480.874,Z 267.806,A -85,B 0,C 180,E1 23362.767,E2 23362.767} C_VEL
LIN {X 0,Y 480.887,Z 267.809,A -85,B 0,C 180,E1 23359.242,E2 23359.242} C_VEL
LIN {X 0,Y 480.857,Z 267.822,A -85,B 0,C 180,E1 23355.665,E2 23355.665} C_VEL
LIN {X 0,Y 480.966,Z 268.32,A -85,B 0,C 180,E1 23355.225,E2 23355.225} C_VEL
LIN {X 0,Y 489.962,Z 287.836,A -85,B 0,C 180,E1 23352.55,E2 23352.55} C_VEL
LIN {X 0,Y 497.252,Z 304.35,A -85,B 0,C 180,E1 23350.53,E2 23350.53} C_VEL
LIN {X 0,Y 499.925,Z 309.249,A -85,B 0,C 180,E1 23350.198,E2 23350.198} C_VEL
LIN {X 0,Y 502.621,Z 326.577,A -85,B 0,C 180,E1 23349.651,E2 23349.651} C_VEL
LIN {X 0,Y 499.038,Z 535.718,A -85,B 0,C 180,E1 23346.28,E2 23346.28} C_VEL
LIN {X 0,Y 497.815,Z 609.272,A -85,B 0,C 180,E1 23345.094,E2 23345.094} C_VEL
LIN {X 0,Y 496.891,Z 630.724,A -85,B 0,C 180,E1 23344.549,E2 23344.549} C_VEL
LIN {X 0,Y 495.658,Z 653.214,A -85,B 0,C 180,E1 23343.761,E2 23343.761} C_VEL
LIN {X 0,Y 494.273,Z 674.575,A -85,B 0,C 180,E1 23342.79,E2 23342.79} C_VEL
LIN {X 0,Y 492.69,Z 694.936,A -85,B 0,C 180,E1 23341.64,E2 23341.64} C_VEL
LIN {X 0,Y 491.077,Z 714.073,A -85,B 0,C 180,E1 23340.326,E2 23340.326} C_VEL
LIN {X 0,Y 489.299,Z 732.094,A -85,B 0,C 180,E1 23338.832,E2 23338.832} C_VEL
LIN {X 0,Y 487.495,Z 749.92,A -85,B 0,C 180,E1 23337.085,E2 23337.085} C_VEL
LIN {X 0,Y 485.802,Z 766.18,A -85,B 0,C 180,E1 23335.216,E2 23335.216} C_VEL
LIN {X 0,Y 484.237,Z 782.024,A -85,B 0,C 180,E1 23333.098,E2 23333.098} C_VEL
LIN {X 0,Y 482.995,Z 795.633,A -85,B 0,C 180,E1 23330.985,E2 23330.985} C_VEL
LIN {X 0,Y 481.967,Z 807.819,A -85,B 0,C 180,E1 23328.756,E2 23328.756} C_VEL
LIN {X 0,Y 481.123,Z 819.528,A -85,B 0,C 180,E1 23326.237,E2 23326.237} C_VEL
LIN {X 0,Y 480.579,Z 828.853,A -85,B 0,C 180,E1 23323.843,E2 23323.843} C_VEL
LIN {X 0,Y 480.225,Z 836.529,A -85,B 0,C 180,E1 23321.408,E2 23321.408} C_VEL
LIN {X 0,Y 480.013,Z 843.146,A -85,B 0,C 180,E1 23318.746,E2 23318.746} C_VEL
LIN {X 0,Y 479.939,Z 847.823,A -85,B 0,C 180,E1 23316.219,E2 23316.219} C_VEL
LIN {X 0,Y 479.907,Z 850.787,A -85,B 0,C 180,E1 23313.703,E2 23313.703} C_VEL
LIN {X 0,Y 479.911,Z 852.304,A -85,B 0,C 180,E1 23311.074,E2 23311.074} C_VEL
LIN {X 0,Y 479.905,Z 852.258,A -85,B 0,C 180,E1 23308.687,E2 23308.687} C_VEL
LIN {X 0,Y 479.908,Z 850.671,A -85,B 0,C 180,E1 23306.177,E2 23306.177} C_VEL
LIN {X 0,Y 479.939,Z 847.633,A -85,B 0,C 180,E1 23303.661,E2 23303.661} C_VEL
LIN {X 0,Y 480.013,Z 843.145,A -85,B 0,C 180,E1 23301.254,E2 23301.254} C_VEL
LIN {X 0,Y 480.211,Z 836.881,A -85,B 0,C 180,E1 23298.714,E2 23298.714} C_VEL
LIN {X 0,Y 480.555,Z 829.258,A -85,B 0,C 180,E1 23296.28,E2 23296.28} C_VEL
LIN {X 0,Y 481.104,Z 819.81,A -85,B 0,C 180,E1 23293.831,E2 23293.831} C_VEL
LIN {X 0,Y 481.92,Z 808.454,A -85,B 0,C 180,E1 23291.367,E2 23291.367} C_VEL
LIN {X 0,Y 482.926,Z 796.352,A -85,B 0,C 180,E1 23289.139,E2 23289.139} C_VEL
LIN {X 0,Y 484.152,Z 782.869,A -85,B 0,C 180,E1 23287.026,E2 23287.026} C_VEL
LIN {X 0,Y 485.754,Z 766.687,A -85,B 0,C 180,E1 23284.847,E2 23284.847} C_VEL
LIN {X 0,Y 487.438,Z 750.525,A -85,B 0,C 180,E1 23282.978,E2 23282.978} C_VEL
LIN {X 0,Y 489.185,Z 733.123,A -85,B 0,C 180,E1 23281.264,E2 23281.264} C_VEL
LIN {X 0,Y 491.004,Z 714.905,A -85,B 0,C 180,E1 23279.736,E2 23279.736} C_VEL
LIN {X 0,Y 492.616,Z 695.987,A -85,B 0,C 180,E1 23278.423,E2 23278.423} C_VEL
LIN {X 0,Y 494.136,Z 676.271,A -85,B 0,C 180,E1 23277.3,E2 23277.3} C_VEL
LIN {X 0,Y 495.574,Z 654.757,A -85,B 0,C 180,E1 23276.302,E2 23276.302} C_VEL
LIN {X 0,Y 496.776,Z 633.295,A -85,B 0,C 180,E1 23275.524,E2 23275.524} C_VEL
LIN {X 0,Y 497.691,Z 612.292,A -85,B 0,C 180,E1 23274.975,E2 23274.975} C_VEL
LIN {X 0,Y 498.344,Z 581.473,A -85,B 0,C 180,E1 23274.441,E2 23274.441} C_VEL
LIN {X 0,Y 501.842,Z 367.807,A -85,B 0,C 180,E1 23271.027,E2 23271.027} C_VEL
LIN {X 0,Y 502.482,Z 324.592,A -85,B 0,C 180,E1 23270.301,E2 23270.301} C_VEL
LIN {X 0,Y 499.585,Z 308.258,A -85,B 0,C 180,E1 23269.753,E2 23269.753} C_VEL
LIN {X 0,Y 496.681,Z 303.289,A -85,B 0,C 180,E1 23269.37,E2 23269.37} C_VEL
LIN {X 0,Y 487.877,Z 283.266,A -85,B 0,C 180,E1 23266.852,E2 23266.852} C_VEL
LIN {X 0,Y 481.953,Z 270.91,A -85,B 0,C 180,E1 23265.143,E2 23265.143} C_VEL
LIN {X 0,Y 480.909,Z 268.015,A -85,B 0,C 180,E1 23264.701,E2 23264.701} C_VEL
LIN {X 0,Y 480.888,Z 267.804,A -85,B 0,C 180,E1 23261.18,E2 23261.18} C_VEL
LIN {X 0,Y 480.846,Z 267.814,A -85,B 0,C 180,E1 23257.686,E2 23257.686} C_VEL
LIN {X 0,Y 480.843,Z 267.84,A -85,B 0,C 180,E1 23254.15,E2 23254.15} C_VEL
LIN {X 0,Y 480.872,Z 267.804,A -85,B 0,C 180,E1 23250.625,E2 23250.625} C_VEL
LIN {X 0,Y 480.871,Z 267.832,A -85,B 0,C 180,E1 23247.088,E2 23247.088} C_VEL
LIN {X 0,Y 480.826,Z 267.835,A -85,B 0,C 180,E1 23243.661,E2 23243.661} C_VEL
LIN {X 0,Y 480.822,Z 267.831,A -85,B 0,C 180,E1 23239.966,E2 23239.966} C_VEL
LIN {X 0,Y 480.858,Z 267.83,A -85,B 0,C 180,E1 23236.551,E2 23236.551} C_VEL
LIN {X 0,Y 480.841,Z 267.84,A -85,B 0,C 180,E1 23233.1,E2 23233.1} C_VEL
LIN {X 0,Y 480.817,Z 267.84,A -85,B 0,C 180,E1 23229.576,E2 23229.576} C_VEL
LIN {X 0,Y 480.829,Z 267.838,A -85,B 0,C 180,E1 23225.968,E2 23225.968} C_VEL
LIN {X 0,Y 480.877,Z 267.827,A -85,B 0,C 180,E1 23222.502,E2 23222.502} C_VEL
LIN {X 0,Y 480.853,Z 267.831,A -85,B 0,C 180,E1 23219.047,E2 23219.047} C_VEL
LIN {X 0,Y 480.834,Z 267.837,A -85,B 0,C 180,E1 23215.587,E2 23215.587} C_VEL
LIN {X 0,Y 480.864,Z 267.835,A -85,B 0,C 180,E1 23212.112,E2 23212.112} C_VEL
LIN {X 0,Y 480.89,Z 267.829,A -85,B 0,C 180,E1 23208.608,E2 23208.608} C_VEL
LIN {X 0,Y 480.861,Z 267.826,A -85,B 0,C 180,E1 23205.058,E2 23205.058} C_VEL
LIN {X 0,Y 480.852,Z 267.827,A -85,B 0,C 180,E1 23201.449,E2 23201.449} C_VEL
LIN {X 0,Y 480.871,Z 267.825,A -85,B 0,C 180,E1 23197.892,E2 23197.892} C_VEL
LIN {X 0,Y 480.892,Z 267.824,A -85,B 0,C 180,E1 23194.375,E2 23194.375} C_VEL
LIN {X 0,Y 480.887,Z 267.822,A -85,B 0,C 180,E1 23190.75,E2 23190.75} C_VEL
LIN {X 0,Y 480.868,Z 267.82,A -85,B 0,C 180,E1 23187.133,E2 23187.133} C_VEL
LIN {X 0,Y 480.871,Z 267.809,A -85,B 0,C 180,E1 23183.511,E2 23183.511} C_VEL
LIN {X 0,Y 480.891,Z 267.833,A -85,B 0,C 180,E1 23179.917,E2 23179.917} C_VEL
LIN {X 0,Y 480.884,Z 267.817,A -85,B 0,C 180,E1 23176.346,E2 23176.346} C_VEL
LIN {X 0,Y 480.885,Z 267.808,A -85,B 0,C 180,E1 23172.672,E2 23172.672} C_VEL
LIN {X 0,Y 480.958,Z 268.322,A -85,B 0,C 180,E1 23172.15,E2 23172.15} C_VEL
LIN {X 0,Y 489.13,Z 287.09,A -85,B 0,C 180,E1 23169.403,E2 23169.403} C_VEL
LIN {X 0,Y 496.327,Z 304.965,A -85,B 0,C 180,E1 23167.036,E2 23167.036} C_VEL
LIN {X 0,Y 494.863,Z 327.535,A -85,B 0,C 180,E1 23165.177,E2 23165.177} C_VEL
LIN {X 0,Y 499.038,Z 351.766,A -85,B 0,C 180,E1 23164.393,E2 23164.393} C_VEL
LIN {X 0,Y 498.975,Z 355.582,A -85,B 0,C 180,E1 23164.334,E2 23164.334} C_VEL
LIN {X 0,Y 498.05,Z 363.281,A -85,B 0,C 180,E1 23164.283,E2 23164.283} C_VEL
LIN {X 0,Y 492.723,Z 383.826,A -85,B 0,C 180,E1 23164.399,E2 23164.399} C_VEL
LIN {X 0,Y 492.018,Z 390.433,A -85,B 0,C 180,E1 23164.349,E2 23164.349} C_VEL
LIN {X 0,Y 488.973,Z 591.873,A -85,B 0,C 180,E1 23161.211,E2 23161.211} C_VEL
LIN {X 0,Y 488.144,Z 611.603,A -85,B 0,C 180,E1 23160.707,E2 23160.707} C_VEL
LIN {X 0,Y 486.91,Z 631.963,A -85,B 0,C 180,E1 23159.967,E2 23159.967} C_VEL
LIN {X 0,Y 485.424,Z 651.566,A -85,B 0,C 180,E1 23159.016,E2 23159.016} C_VEL
LIN {X 0,Y 483.799,Z 669.726,A -85,B 0,C 180,E1 23157.91,E2 23157.91} C_VEL
LIN {X 0,Y 481.963,Z 687.786,A -85,B 0,C 180,E1 23156.555,E2 23156.555} C_VEL
LIN {X 0,Y 480.087,Z 704.799,A -85,B 0,C 180,E1 23155.009,E2 23155.009} C_VEL
LIN {X 0,Y 478.264,Z 720.892,A -85,B 0,C 180,E1 23153.273,E2 23153.273} C_VEL
LIN {X 0,Y 476.598,Z 736.008,A -85,B 0,C 180,E1 23151.334,E2 23151.334} C_VEL
LIN {X 0,Y 475.177,Z 749.47,A -85,B 0,C 180,E1 23149.29,E2 23149.29} C_VEL
LIN {X 0,Y 474.005,Z 761.903,A -85,B 0,C 180,E1 23147.049,E2 23147.049} C_VEL
LIN {X 0,Y 473.161,Z 772.306,A -85,B 0,C 180,E1 23144.814,E2 23144.814} C_VEL
LIN {X 0,Y 472.529,Z 781.719,A -85,B 0,C 180,E1 23142.34,E2 23142.34} C_VEL
LIN {X 0,Y 472.171,Z 789.161,A -85,B 0,C 180,E1 23139.876,E2 23139.876} C_VEL
LIN {X 0,Y 471.992,Z 795.16,A -85,B 0,C 180,E1 23137.302,E2 23137.302} C_VEL
LIN {X 0,Y 471.928,Z 799.207,A -85,B 0,C 180,E1 23134.861,E2 23134.861} C_VEL
LIN {X 0,Y 471.909,Z 801.639,A -85,B 0,C 180,E1 23132.429,E2 23132.429} C_VEL
LIN {X 0,Y 471.914,Z 802.494,A -85,B 0,C 180,E1 23130,E2 23130} C_VEL
LIN {X 0,Y 471.905,Z 801.692,A -85,B 0,C 180,E1 23127.571,E2 23127.571} C_VEL
LIN {X 0,Y 471.928,Z 799.325,A -85,B 0,C 180,E1 23125.139,E2 23125.139} C_VEL
LIN {X 0,Y 471.989,Z 795.346,A -85,B 0,C 180,E1 23122.698,E2 23122.698} C_VEL
LIN {X 0,Y 472.163,Z 789.412,A -85,B 0,C 180,E1 23120.124,E2 23120.124} C_VEL
LIN {X 0,Y 472.512,Z 782.036,A -85,B 0,C 180,E1 23117.66,E2 23117.66} C_VEL
LIN {X 0,Y 473.13,Z 772.666,A -85,B 0,C 180,E1 23115.185,E2 23115.185} C_VEL
LIN {X 0,Y 474.006,Z 761.865,A -85,B 0,C 180,E1 23112.853,E2 23112.853} C_VEL
LIN {X 0,Y 475.122,Z 749.989,A -85,B 0,C 180,E1 23110.708,E2 23110.708} C_VEL
LIN {X 0,Y 476.582,Z 736.101,A -85,B 0,C 180,E1 23108.59,E2 23108.59} C_VEL
LIN {X 0,Y 478.245,Z 721.091,A -85,B 0,C 180,E1 23106.661,E2 23106.661} C_VEL
LIN {X 0,Y 480.015,Z 705.53,A -85,B 0,C 180,E1 23104.971,E2 23104.971} C_VEL
LIN {X 0,Y 481.889,Z 688.536,A -85,B 0,C 180,E1 23103.415,E2 23103.415} C_VEL
LIN {X 0,Y 483.681,Z 670.89,A -85,B 0,C 180,E1 23102.082,E2 23102.082} C_VEL
LIN {X 0,Y 485.292,Z 653.04,A -85,B 0,C 180,E1 23100.975,E2 23100.975} C_VEL
LIN {X 0,Y 486.836,Z 633.161,A -85,B 0,C 180,E1 23099.994,E2 23099.994} C_VEL
LIN {X 0,Y 488.048,Z 613.549,A -85,B 0,C 180,E1 23099.261,E2 23099.261} C_VEL
LIN {X 0,Y 488.942,Z 593.274,A -85,B 0,C 180,E1 23098.726,E2 23098.726} C_VEL
LIN {X 0,Y 490.225,Z 512.836,A -85,B 0,C 180,E1 23097.453,E2 23097.453} C_VEL
LIN {X 0,Y 492.496,Z 351.433,A -85,B 0,C 180,E1 23094.934,E2 23094.934} C_VEL
LIN {X 0,Y 488.143,Z 326.405,A -85,B 0,C 180,E1 23094.068,E2 23094.068} C_VEL
LIN {X 0,Y 489.329,Z 307.956,A -85,B 0,C 180,E1 23092.49,E2 23092.49} C_VEL
LIN {X 0,Y 482.03,Z 289.853,A -85,B 0,C 180,E1 23090.036,E2 23090.036} C_VEL
LIN {X 0,Y 475.664,Z 275.517,A -85,B 0,C 180,E1 23087.904,E2 23087.904} C_VEL
LIN {X 0,Y 472.98,Z 269.057,A -85,B 0,C 180,E1 23086.872,E2 23086.872} C_VEL
LIN {X 0,Y 472.945,Z 268.8,A -85,B 0,C 180,E1 23083.345,E2 23083.345} C_VEL
LIN {X 0,Y 472.945,Z 268.825,A -85,B 0,C 180,E1 23079.677,E2 23079.677} C_VEL
LIN {X 0,Y 472.948,Z 268.801,A -85,B 0,C 180,E1 23075.996,E2 23075.996} C_VEL
LIN {X 0,Y 472.936,Z 268.797,A -85,B 0,C 180,E1 23072.336,E2 23072.336} C_VEL
LIN {X 0,Y 472.931,Z 268.824,A -85,B 0,C 180,E1 23068.675,E2 23068.675} C_VEL
LIN {X 0,Y 472.938,Z 268.823,A -85,B 0,C 180,E1 23065.014,E2 23065.014} C_VEL
LIN {X 0,Y 472.954,Z 268.816,A -85,B 0,C 180,E1 23061.453,E2 23061.453} C_VEL
LIN {X 0,Y 472.945,Z 268.813,A -85,B 0,C 180,E1 23057.851,E2 23057.851} C_VEL
LIN {X 0,Y 472.915,Z 268.814,A -85,B 0,C 180,E1 23054.322,E2 23054.322} C_VEL
LIN {X 0,Y 472.91,Z 268.812,A -85,B 0,C 180,E1 23050.6,E2 23050.6} C_VEL
LIN {X 0,Y 472.931,Z 268.818,A -85,B 0,C 180,E1 23047.044,E2 23047.044} C_VEL
LIN {X 0,Y 472.95,Z 268.826,A -85,B 0,C 180,E1 23043.394,E2 23043.394} C_VEL
LIN {X 0,Y 472.912,Z 268.823,A -85,B 0,C 180,E1 23039.879,E2 23039.879} C_VEL
LIN {X 0,Y 472.889,Z 268.823,A -85,B 0,C 180,E1 23036.331,E2 23036.331} C_VEL
LIN {X 0,Y 472.903,Z 268.817,A -85,B 0,C 180,E1 23032.834,E2 23032.834} C_VEL
LIN {X 0,Y 472.933,Z 268.816,A -85,B 0,C 180,E1 23029.278,E2 23029.278} C_VEL
LIN {X 0,Y 472.889,Z 268.828,A -85,B 0,C 180,E1 23025.803,E2 23025.803} C_VEL
LIN {X 0,Y 472.875,Z 268.828,A -85,B 0,C 180,E1 23022.274,E2 23022.274} C_VEL
LIN {X 0,Y 472.896,Z 268.827,A -85,B 0,C 180,E1 23018.675,E2 23018.675} C_VEL
LIN {X 0,Y 472.938,Z 268.826,A -85,B 0,C 180,E1 23015.254,E2 23015.254} C_VEL
LIN {X 0,Y 472.903,Z 268.829,A -85,B 0,C 180,E1 23011.732,E2 23011.732} C_VEL
LIN {X 0,Y 472.892,Z 268.794,A -85,B 0,C 180,E1 23008.206,E2 23008.206} C_VEL
LIN {X 0,Y 472.925,Z 268.814,A -85,B 0,C 180,E1 23004.692,E2 23004.692} C_VEL
LIN {X 0,Y 472.96,Z 268.821,A -85,B 0,C 180,E1 23001.073,E2 23001.073} C_VEL
LIN {X 0,Y 472.922,Z 268.801,A -85,B 0,C 180,E1 22997.548,E2 22997.548} C_VEL
LIN {X 0,Y 472.958,Z 269.14,A -85,B 0,C 180,E1 22996.1,E2 22996.1} C_VEL
LIN {X 0,Y 474.347,Z 272.476,A -85,B 0,C 180,E1 22995.589,E2 22995.589} C_VEL
LIN {X 0,Y 481.992,Z 288.492,A -85,B 0,C 180,E1 22993.319,E2 22993.319} C_VEL
LIN {X 0,Y 489.086,Z 304.658,A -85,B 0,C 180,E1 22991.276,E2 22991.276} C_VEL
LIN {X 0,Y 493.953,Z 313.154,A -85,B 0,C 180,E1 22990.661,E2 22990.661} C_VEL
LIN {X 0,Y 496.207,Z 328.072,A -85,B 0,C 180,E1 22990.183,E2 22990.183} C_VEL
LIN {X 0,Y 492.23,Z 538.766,A -85,B 0,C 180,E1 22986.729,E2 22986.729} C_VEL
LIN {X 0,Y 490.95,Z 608.999,A -85,B 0,C 180,E1 22985.578,E2 22985.578} C_VEL
LIN {X 0,Y 489.971,Z 630.427,A -85,B 0,C 180,E1 22985.027,E2 22985.027} C_VEL
LIN {X 0,Y 488.665,Z 652.678,A -85,B 0,C 180,E1 22984.24,E2 22984.24} C_VEL
LIN {X 0,Y 487.238,Z 673.422,A -85,B 0,C 180,E1 22983.293,E2 22983.293} C_VEL
LIN {X 0,Y 485.592,Z 693.4,A -85,B 0,C 180,E1 22982.158,E2 22982.158} C_VEL
LIN {X 0,Y 483.856,Z 712.792,A -85,B 0,C 180,E1 22980.828,E2 22980.828} C_VEL
LIN {X 0,Y 482.06,Z 731.599,A -85,B 0,C 180,E1 22979.307,E2 22979.307} C_VEL
LIN {X 0,Y 480.549,Z 746.263,A -85,B 0,C 180,E1 22977.913,E2 22977.913} C_VEL
LIN {X 0,Y 478.701,Z 763.138,A -85,B 0,C 180,E1 22976.015,E2 22976.015} C_VEL
LIN {X 0,Y 477.008,Z 778.88,A -85,B 0,C 180,E1 22973.95,E2 22973.95} C_VEL
LIN {X 0,Y 475.508,Z 793.323,A -85,B 0,C 180,E1 22971.72,E2 22971.72} C_VEL
LIN {X 0,Y 474.28,Z 806.547,A -85,B 0,C 180,E1 22969.328,E2 22969.328} C_VEL
LIN {X 0,Y 473.362,Z 817.965,A -85,B 0,C 180,E1 22966.894,E2 22966.894} C_VEL
LIN {X 0,Y 472.718,Z 827.512,A -85,B 0,C 180,E1 22964.453,E2 22964.453} C_VEL
LIN {X 0,Y 472.306,Z 835.469,A -85,B 0,C 180,E1 22961.973,E2 22961.973} C_VEL
LIN {X 0,Y 472.075,Z 842.129,A -85,B 0,C 180,E1 22959.386,E2 22959.386} C_VEL
LIN {X 0,Y 471.964,Z 846.813,A -85,B 0,C 180,E1 22956.935,E2 22956.935} C_VEL
LIN {X 0,Y 471.916,Z 850.332,A -85,B 0,C 180,E1 22954.253,E2 22954.253} C_VEL
LIN {X 0,Y 471.902,Z 852.085,A -85,B 0,C 180,E1 22951.821,E2 22951.821} C_VEL
LIN {X 0,Y 471.902,Z 852.372,A -85,B 0,C 180,E1 22949.272,E2 22949.272} C_VEL
LIN {X 0,Y 471.915,Z 851.235,A -85,B 0,C 180,E1 22946.721,E2 22946.721} C_VEL
LIN {X 0,Y 471.933,Z 848.458,A -85,B 0,C 180,E1 22944.163,E2 22944.163} C_VEL
LIN {X 0,Y 472.013,Z 843.907,A -85,B 0,C 180,E1 22941.473,E2 22941.473} C_VEL
LIN {X 0,Y 472.193,Z 838.249,A -85,B 0,C 180,E1 22939.014,E2 22939.014} C_VEL
LIN {X 0,Y 472.525,Z 830.882,A -85,B 0,C 180,E1 22936.541,E2 22936.541} C_VEL
LIN {X 0,Y 473.119,Z 821.353,A -85,B 0,C 180,E1 22933.928,E2 22933.928} C_VEL
LIN {X 0,Y 473.974,Z 810.354,A -85,B 0,C 180,E1 22931.426,E2 22931.426} C_VEL
LIN {X 0,Y 475.082,Z 797.759,A -85,B 0,C 180,E1 22929.037,E2 22929.037} C_VEL
LIN {X 0,Y 476.474,Z 783.712,A -85,B 0,C 180,E1 22926.765,E2 22926.765} C_VEL
LIN {X 0,Y 478.088,Z 768.713,A -85,B 0,C 180,E1 22924.68,E2 22924.68} C_VEL
LIN {X 0,Y 479.922,Z 752.245,A -85,B 0,C 180,E1 22922.721,E2 22922.721} C_VEL
LIN {X 0,Y 481.493,Z 737.158,A -85,B 0,C 180,E1 22921.2,E2 22921.2} C_VEL
LIN {X 0,Y 483.334,Z 718.659,A -85,B 0,C 180,E1 22919.613,E2 22919.613} C_VEL
LIN {X 0,Y 485.074,Z 699.309,A -85,B 0,C 180,E1 22918.222,E2 22918.222} C_VEL
LIN {X 0,Y 486.807,Z 678.641,A -85,B 0,C 180,E1 22916.987,E2 22916.987} C_VEL
LIN {X 0,Y 488.354,Z 658.008,A -85,B 0,C 180,E1 22915.981,E2 22915.981} C_VEL
LIN {X 0,Y 489.63,Z 636.678,A -85,B 0,C 180,E1 22915.166,E2 22915.166} C_VEL
LIN {X 0,Y 490.686,Z 615.049,A -85,B 0,C 180,E1 22914.562,E2 22914.562} C_VEL
LIN {X 0,Y 491.404,Z 589.832,A -85,B 0,C 180,E1 22914.086,E2 22914.086} C_VEL
LIN {X 0,Y 495.037,Z 386.347,A -85,B 0,C 180,E1 22910.787,E2 22910.787} C_VEL
LIN {X 0,Y 496.059,Z 325.96,A -85,B 0,C 180,E1 22909.765,E2 22909.765} C_VEL
LIN {X 0,Y 493.591,Z 312.186,A -85,B 0,C 180,E1 22909.288,E2 22909.288} C_VEL
LIN {X 0,Y 488.527,Z 303.565,A -85,B 0,C 180,E1 22908.619,E2 22908.619} C_VEL
LIN {X 0,Y 480.463,Z 285.142,A -85,B 0,C 180,E1 22906.229,E2 22906.229} C_VEL
LIN {X 0,Y 474.182,Z 272.228,A -85,B 0,C 180,E1 22904.374,E2 22904.374} C_VEL
LIN {X 0,Y 472.941,Z 269.026,A -85,B 0,C 180,E1 22903.871,E2 22903.871} C_VEL
LIN {X 0,Y 472.922,Z 268.804,A -85,B 0,C 180,E1 22900.439,E2 22900.439} C_VEL
LIN {X 0,Y 472.951,Z 268.789,A -85,B 0,C 180,E1 22896.898,E2 22896.898} C_VEL
LIN {X 0,Y 472.921,Z 268.821,A -85,B 0,C 180,E1 22893.346,E2 22893.346} C_VEL
LIN {X 0,Y 472.893,Z 268.812,A -85,B 0,C 180,E1 22889.793,E2 22889.793} C_VEL
LIN {X 0,Y 472.899,Z 268.822,A -85,B 0,C 180,E1 22886.224,E2 22886.224} C_VEL
LIN {X 0,Y 472.948,Z 268.814,A -85,B 0,C 180,E1 22882.76,E2 22882.76} C_VEL
LIN {X 0,Y 472.899,Z 268.817,A -85,B 0,C 180,E1 22879.258,E2 22879.258} C_VEL
LIN {X 0,Y 472.873,Z 268.818,A -85,B 0,C 180,E1 22875.703,E2 22875.703} C_VEL
LIN {X 0,Y 472.89,Z 268.819,A -85,B 0,C 180,E1 22872.206,E2 22872.206} C_VEL
LIN {X 0,Y 472.938,Z 268.821,A -85,B 0,C 180,E1 22868.633,E2 22868.633} C_VEL
LIN {X 0,Y 472.907,Z 268.828,A -85,B 0,C 180,E1 22865.094,E2 22865.094} C_VEL
LIN {X 0,Y 472.888,Z 268.825,A -85,B 0,C 180,E1 22861.575,E2 22861.575} C_VEL
LIN {X 0,Y 472.909,Z 268.818,A -85,B 0,C 180,E1 22858.061,E2 22858.061} C_VEL
LIN {X 0,Y 472.95,Z 268.811,A -85,B 0,C 180,E1 22854.541,E2 22854.541} C_VEL
LIN {X 0,Y 472.923,Z 268.824,A -85,B 0,C 180,E1 22850.999,E2 22850.999} C_VEL
LIN {X 0,Y 472.905,Z 268.826,A -85,B 0,C 180,E1 22847.422,E2 22847.422} C_VEL
LIN {X 0,Y 472.919,Z 268.824,A -85,B 0,C 180,E1 22843.795,E2 22843.795} C_VEL
LIN {X 0,Y 472.95,Z 268.822,A -85,B 0,C 180,E1 22840.177,E2 22840.177} C_VEL
LIN {X 0,Y 472.954,Z 268.818,A -85,B 0,C 180,E1 22836.56,E2 22836.56} C_VEL
LIN {X 0,Y 472.942,Z 268.818,A -85,B 0,C 180,E1 22832.876,E2 22832.876} C_VEL
LIN {X 0,Y 472.924,Z 268.791,A -85,B 0,C 180,E1 22829.368,E2 22829.368} C_VEL
LIN {X 0,Y 472.943,Z 268.823,A -85,B 0,C 180,E1 22825.751,E2 22825.751} C_VEL
LIN {X 0,Y 472.949,Z 268.792,A -85,B 0,C 180,E1 22822.049,E2 22822.049} C_VEL
LIN {X 0,Y 472.946,Z 268.794,A -85,B 0,C 180,E1 22818.407,E2 22818.407} C_VEL
LIN {X 0,Y 472.948,Z 268.811,A -85,B 0,C 180,E1 22814.737,E2 22814.737} C_VEL
LIN {X 0,Y 472.975,Z 269.045,A -85,B 0,C 180,E1 22813.035,E2 22813.035} C_VEL
LIN {X 0,Y 474.366,Z 272.484,A -85,B 0,C 180,E1 22812.462,E2 22812.462} C_VEL
LIN {X 0,Y 481.634,Z 288.949,A -85,B 0,C 180,E1 22810.001,E2 22810.001} C_VEL
LIN {X 0,Y 489.062,Z 307.242,A -85,B 0,C 180,E1 22807.51,E2 22807.51} C_VEL
LIN {X 0,Y 489.481,Z 308.556,A -85,B 0,C 180,E1 22807.349,E2 22807.349} C_VEL
LIN {X 0,Y 488.193,Z 327.322,A -85,B 0,C 180,E1 22805.789,E2 22805.789} C_VEL
LIN {X 0,Y 492.633,Z 353.211,A -85,B 0,C 180,E1 22804.931,E2 22804.931} C_VEL
LIN {X 0,Y 492.018,Z 390.433,A -85,B 0,C 180,E1 22804.349,E2 22804.349} C_VEL
LIN {X 0,Y 491.102,Z 398.133,A -85,B 0,C 180,E1 22804.298,E2 22804.298} C_VEL
LIN {X 0,Y 485.781,Z 418.681,A -85,B 0,C 180,E1 22804.419,E2 22804.419} C_VEL
LIN {X 0,Y 485.069,Z 425.29,A -85,B 0,C 180,E1 22804.37,E2 22804.37} C_VEL
LIN {X 0,Y 482.413,Z 593.123,A -85,B 0,C 180,E1 22801.736,E2 22801.736} C_VEL
LIN {X 0,Y 481.521,Z 613.103,A -85,B 0,C 180,E1 22801.215,E2 22801.215} C_VEL
LIN {X 0,Y 480.264,Z 632.85,A -85,B 0,C 180,E1 22800.484,E2 22800.484} C_VEL
LIN {X 0,Y 478.716,Z 652.309,A -85,B 0,C 180,E1 22799.531,E2 22799.531} C_VEL
LIN {X 0,Y 476.978,Z 670.435,A -85,B 0,C 180,E1 22798.414,E2 22798.414} C_VEL
LIN {X 0,Y 475.02,Z 688.469,A -85,B 0,C 180,E1 22797.042,E2 22797.042} C_VEL
LIN {X 0,Y 473.016,Z 705.226,A -85,B 0,C 180,E1 22795.499,E2 22795.499} C_VEL
LIN {X 0,Y 471.083,Z 720.907,A -85,B 0,C 180,E1 22793.782,E2 22793.782} C_VEL
LIN {X 0,Y 469.201,Z 736.406,A -85,B 0,C 180,E1 22791.764,E2 22791.764} C_VEL
LIN {X 0,Y 467.592,Z 750.295,A -85,B 0,C 180,E1 22789.615,E2 22789.615} C_VEL
LIN {X 0,Y 466.341,Z 762.209,A -85,B 0,C 180,E1 22787.426,E2 22787.426} C_VEL
LIN {X 0,Y 465.357,Z 772.935,A -85,B 0,C 180,E1 22785.068,E2 22785.068} C_VEL
LIN {X 0,Y 464.652,Z 782.3,A -85,B 0,C 180,E1 22782.552,E2 22782.552} C_VEL
LIN {X 0,Y 464.239,Z 789.696,A -85,B 0,C 180,E1 22780.047,E2 22780.047} C_VEL
LIN {X 0,Y 464.025,Z 795.329,A -85,B 0,C 180,E1 22777.553,E2 22777.553} C_VEL
LIN {X 0,Y 463.939,Z 799.474,A -85,B 0,C 180,E1 22774.945,E2 22774.945} C_VEL
LIN {X 0,Y 463.911,Z 801.888,A -85,B 0,C 180,E1 22772.347,E2 22772.347} C_VEL
LIN {X 0,Y 463.915,Z 802.645,A -85,B 0,C 180,E1 22769.877,E2 22769.877} C_VEL
LIN {X 0,Y 463.908,Z 801.807,A -85,B 0,C 180,E1 22767.406,E2 22767.406} C_VEL
LIN {X 0,Y 463.938,Z 799.43,A -85,B 0,C 180,E1 22764.931,E2 22764.931} C_VEL
LIN {X 0,Y 464.026,Z 795.255,A -85,B 0,C 180,E1 22762.323,E2 22762.323} C_VEL
LIN {X 0,Y 464.245,Z 789.598,A -85,B 0,C 180,E1 22759.828,E2 22759.828} C_VEL
LIN {X 0,Y 464.661,Z 782.177,A -85,B 0,C 180,E1 22757.322,E2 22757.322} C_VEL
LIN {X 0,Y 465.374,Z 772.789,A -85,B 0,C 180,E1 22754.805,E2 22754.805} C_VEL
LIN {X 0,Y 466.383,Z 761.827,A -85,B 0,C 180,E1 22752.406,E2 22752.406} C_VEL
LIN {X 0,Y 467.678,Z 749.546,A -85,B 0,C 180,E1 22750.167,E2 22750.167} C_VEL
LIN {X 0,Y 469.235,Z 736.127,A -85,B 0,C 180,E1 22748.106,E2 22748.106} C_VEL
LIN {X 0,Y 471.012,Z 721.471,A -85,B 0,C 180,E1 22746.195,E2 22746.195} C_VEL
LIN {X 0,Y 472.97,Z 705.656,A -85,B 0,C 180,E1 22744.453,E2 22744.453} C_VEL
LIN {X 0,Y 474.983,Z 688.804,A -85,B 0,C 180,E1 22742.895,E2 22742.895} C_VEL
LIN {X 0,Y 476.951,Z 670.713,A -85,B 0,C 180,E1 22741.516,E2 22741.516} C_VEL
LIN {X 0,Y 478.684,Z 652.657,A -85,B 0,C 180,E1 22740.398,E2 22740.398} C_VEL
LIN {X 0,Y 480.248,Z 633.089,A -85,B 0,C 180,E1 22739.436,E2 22739.436} C_VEL
LIN {X 0,Y 481.519,Z 613.169,A -85,B 0,C 180,E1 22738.698,E2 22738.698} C_VEL
LIN {X 0,Y 482.415,Z 593.151,A -85,B 0,C 180,E1 22738.174,E2 22738.174} C_VEL
LIN {X 0,Y 485.142,Z 421.288,A -85,B 0,C 180,E1 22735.476,E2 22735.476} C_VEL
LIN {X 0,Y 486.127,Z 352.747,A -85,B 0,C 180,E1 22734.376,E2 22734.376} C_VEL
LIN {X 0,Y 481.533,Z 326.263,A -85,B 0,C 180,E1 22733.444,E2 22733.444} C_VEL
LIN {X 0,Y 482.581,Z 311.537,A -85,B 0,C 180,E1 22732.174,E2 22732.174} C_VEL
LIN {X 0,Y 475.109,Z 292.893,A -85,B 0,C 180,E1 22729.597,E2 22729.597} C_VEL
LIN {X 0,Y 467.922,Z 276.818,A -85,B 0,C 180,E1 22727.132,E2 22727.132} C_VEL
LIN {X 0,Y 465.038,Z 270.029,A -85,B 0,C 180,E1 22726.001,E2 22726.001} C_VEL
LIN {X 0,Y 465.004,Z 269.777,A -85,B 0,C 180,E1 22722.468,E2 22722.468} C_VEL
LIN {X 0,Y 465.002,Z 269.801,A -85,B 0,C 180,E1 22718.889,E2 22718.889} C_VEL
LIN {X 0,Y 465.008,Z 269.803,A -85,B 0,C 180,E1 22715.188,E2 22715.188} C_VEL
LIN {X 0,Y 465.009,Z 269.772,A -85,B 0,C 180,E1 22711.5,E2 22711.5} C_VEL
LIN {X 0,Y 465.017,Z 269.811,A -85,B 0,C 180,E1 22707.813,E2 22707.813} C_VEL
LIN {X 0,Y 465,Z 269.812,A -85,B 0,C 180,E1 22704.114,E2 22704.114} C_VEL
LIN {X 0,Y 464.982,Z 269.814,A -85,B 0,C 180,E1 22700.518,E2 22700.518} C_VEL
LIN {X 0,Y 464.988,Z 269.816,A -85,B 0,C 180,E1 22696.876,E2 22696.876} C_VEL
LIN {X 0,Y 465.013,Z 269.805,A -85,B 0,C 180,E1 22693.301,E2 22693.301} C_VEL
LIN {X 0,Y 465.005,Z 269.798,A -85,B 0,C 180,E1 22689.655,E2 22689.655} C_VEL
LIN {X 0,Y 464.969,Z 269.803,A -85,B 0,C 180,E1 22686.173,E2 22686.173} C_VEL
LIN {X 0,Y 464.96,Z 269.81,A -85,B 0,C 180,E1 22682.465,E2 22682.465} C_VEL
LIN {X 0,Y 464.975,Z 269.814,A -85,B 0,C 180,E1 22678.891,E2 22678.891} C_VEL
LIN {X 0,Y 465.002,Z 269.812,A -85,B 0,C 180,E1 22675.313,E2 22675.313} C_VEL
LIN {X 0,Y 464.96,Z 269.808,A -85,B 0,C 180,E1 22671.841,E2 22671.841} C_VEL
LIN {X 0,Y 464.939,Z 269.806,A -85,B 0,C 180,E1 22668.338,E2 22668.338} C_VEL
LIN {X 0,Y 464.955,Z 269.805,A -85,B 0,C 180,E1 22664.79,E2 22664.79} C_VEL
LIN {X 0,Y 464.99,Z 269.804,A -85,B 0,C 180,E1 22661.184,E2 22661.184} C_VEL
LIN {X 0,Y 464.966,Z 269.811,A -85,B 0,C 180,E1 22657.614,E2 22657.614} C_VEL
LIN {X 0,Y 464.95,Z 269.814,A -85,B 0,C 180,E1 22654.117,E2 22654.117} C_VEL
LIN {X 0,Y 464.965,Z 269.805,A -85,B 0,C 180,E1 22650.499,E2 22650.499} C_VEL
LIN {X 0,Y 465.007,Z 269.797,A -85,B 0,C 180,E1 22646.988,E2 22646.988} C_VEL
LIN {X 0,Y 464.995,Z 269.779,A -85,B 0,C 180,E1 22643.324,E2 22643.324} C_VEL
LIN {X 0,Y 464.969,Z 269.799,A -85,B 0,C 180,E1 22639.826,E2 22639.826} C_VEL
LIN {X 0,Y 465.052,Z 270.059,A -85,B 0,C 180,E1 22636.995,E2 22636.995} C_VEL
LIN {X 0,Y 466.496,Z 273.6,A -85,B 0,C 180,E1 22636.421,E2 22636.421} C_VEL
LIN {X 0,Y 473.086,Z 287.314,A -85,B 0,C 180,E1 22634.39,E2 22634.39} C_VEL
LIN {X 0,Y 480.85,Z 304.678,A -85,B 0,C 180,E1 22632.07,E2 22632.07} C_VEL
LIN {X 0,Y 488,Z 316.97,A -85,B 0,C 180,E1 22631.137,E2 22631.137} C_VEL
LIN {X 0,Y 489.829,Z 329.534,A -85,B 0,C 180,E1 22630.729,E2 22630.729} C_VEL
LIN {X 0,Y 485.472,Z 541.118,A -85,B 0,C 180,E1 22627.204,E2 22627.204} C_VEL
LIN {X 0,Y 484.086,Z 608.968,A -85,B 0,C 180,E1 22626.065,E2 22626.065} C_VEL
LIN {X 0,Y 483.049,Z 630.444,A -85,B 0,C 180,E1 22625.506,E2 22625.506} C_VEL
LIN {X 0,Y 481.674,Z 652.548,A -85,B 0,C 180,E1 22624.713,E2 22624.713} C_VEL
LIN {X 0,Y 480.186,Z 672.918,A -85,B 0,C 180,E1 22623.776,E2 22623.776} C_VEL
LIN {X 0,Y 478.452,Z 692.912,A -85,B 0,C 180,E1 22622.626,E2 22622.626} C_VEL
LIN {X 0,Y 476.59,Z 712.322,A -85,B 0,C 180,E1 22621.28,E2 22621.28} C_VEL
LIN {X 0,Y 474.69,Z 731.151,A -85,B 0,C 180,E1 22619.738,E2 22619.738} C_VEL
LIN {X 0,Y 472.763,Z 749.08,A -85,B 0,C 180,E1 22618.002,E2 22618.002} C_VEL
LIN {X 0,Y 470.932,Z 765.895,A -85,B 0,C 180,E1 22616.092,E2 22616.092} C_VEL
LIN {X 0,Y 469.397,Z 779.557,A -85,B 0,C 180,E1 22614.262,E2 22614.262} C_VEL
LIN {X 0,Y 467.847,Z 793.321,A -85,B 0,C 180,E1 22612.094,E2 22612.094} C_VEL
LIN {X 0,Y 466.512,Z 806.546,A -85,B 0,C 180,E1 22609.663,E2 22609.663} C_VEL
LIN {X 0,Y 465.531,Z 817.749,A -85,B 0,C 180,E1 22607.241,E2 22607.241} C_VEL
LIN {X 0,Y 464.805,Z 827.512,A -85,B 0,C 180,E1 22604.704,E2 22604.704} C_VEL
LIN {X 0,Y 464.343,Z 835.544,A -85,B 0,C 180,E1 22602.155,E2 22602.155} C_VEL
LIN {X 0,Y 464.088,Z 842.129,A -85,B 0,C 180,E1 22599.549,E2 22599.549} C_VEL
LIN {X 0,Y 463.971,Z 846.813,A -85,B 0,C 180,E1 22597.056,E2 22597.056} C_VEL
LIN {X 0,Y 463.918,Z 850.332,A -85,B 0,C 180,E1 22594.326,E2 22594.326} C_VEL
LIN {X 0,Y 463.903,Z 852.085,A -85,B 0,C 180,E1 22591.853,E2 22591.853} C_VEL
LIN {X 0,Y 463.903,Z 852.371,A -85,B 0,C 180,E1 22589.259,E2 22589.259} C_VEL
LIN {X 0,Y 463.914,Z 851.235,A -85,B 0,C 180,E1 22586.664,E2 22586.664} C_VEL
LIN {X 0,Y 463.934,Z 848.617,A -85,B 0,C 180,E1 22584.187,E2 22584.187} C_VEL
LIN {X 0,Y 464.02,Z 844.161,A -85,B 0,C 180,E1 22581.45,E2 22581.45} C_VEL
LIN {X 0,Y 464.21,Z 838.553,A -85,B 0,C 180,E1 22578.949,E2 22578.949} C_VEL
LIN {X 0,Y 464.569,Z 831.286,A -85,B 0,C 180,E1 22576.433,E2 22576.433} C_VEL
LIN {X 0,Y 465.17,Z 822.38,A -85,B 0,C 180,E1 22573.903,E2 22573.903} C_VEL
LIN {X 0,Y 466.065,Z 811.52,A -85,B 0,C 180,E1 22571.359,E2 22571.359} C_VEL
LIN {X 0,Y 467.166,Z 799.859,A -85,B 0,C 180,E1 22569.059,E2 22569.059} C_VEL
LIN {X 0,Y 468.625,Z 786.246,A -85,B 0,C 180,E1 22566.752,E2 22566.752} C_VEL
LIN {X 0,Y 470.364,Z 771.168,A -85,B 0,C 180,E1 22564.572,E2 22564.572} C_VEL
LIN {X 0,Y 472.047,Z 755.593,A -85,B 0,C 180,E1 22562.706,E2 22562.706} C_VEL
LIN {X 0,Y 474.001,Z 737.445,A -85,B 0,C 180,E1 22560.843,E2 22560.843} C_VEL
LIN {X 0,Y 475.971,Z 718.914,A -85,B 0,C 180,E1 22559.224,E2 22559.224} C_VEL
LIN {X 0,Y 477.798,Z 699.765,A -85,B 0,C 180,E1 22557.821,E2 22557.821} C_VEL
LIN {X 0,Y 479.685,Z 678.784,A -85,B 0,C 180,E1 22556.543,E2 22556.543} C_VEL
LIN {X 0,Y 481.309,Z 658.401,A -85,B 0,C 180,E1 22555.531,E2 22555.531} C_VEL
LIN {X 0,Y 482.703,Z 636.368,A -85,B 0,C 180,E1 22554.681,E2 22554.681} C_VEL
LIN {X 0,Y 483.811,Z 614.999,A -85,B 0,C 180,E1 22554.077,E2 22554.077} C_VEL
LIN {X 0,Y 484.563,Z 590.83,A -85,B 0,C 180,E1 22553.609,E2 22553.609} C_VEL
LIN {X 0,Y 488.708,Z 381.609,A -85,B 0,C 180,E1 22550.15,E2 22550.15} C_VEL
LIN {X 0,Y 489.682,Z 327.348,A -85,B 0,C 180,E1 22549.216,E2 22549.216} C_VEL
LIN {X 0,Y 487.72,Z 316.154,A -85,B 0,C 180,E1 22548.821,E2 22548.821} C_VEL
LIN {X 0,Y 480.581,Z 304.114,A -85,B 0,C 180,E1 22547.877,E2 22547.877} C_VEL
LIN {X 0,Y 472.662,Z 286.252,A -85,B 0,C 180,E1 22545.47,E2 22545.47} C_VEL
LIN {X 0,Y 466.453,Z 273.536,A -85,B 0,C 180,E1 22543.573,E2 22543.573} C_VEL
LIN {X 0,Y 465.047,Z 270.023,A -85,B 0,C 180,E1 22543,E2 22543} C_VEL
LIN {X 0,Y 464.974,Z 269.813,A -85,B 0,C 180,E1 22539.664,E2 22539.664} C_VEL
LIN {X 0,Y 464.963,Z 269.788,A -85,B 0,C 180,E1 22536.048,E2 22536.048} C_VEL
LIN {X 0,Y 464.984,Z 269.788,A -85,B 0,C 180,E1 22532.519,E2 22532.519} C_VEL
LIN {X 0,Y 465.012,Z 269.805,A -85,B 0,C 180,E1 22528.933,E2 22528.933} C_VEL
LIN {X 0,Y 464.966,Z 269.814,A -85,B 0,C 180,E1 22525.336,E2 22525.336} C_VEL
LIN {X 0,Y 464.945,Z 269.816,A -85,B 0,C 180,E1 22521.841,E2 22521.841} C_VEL
LIN {X 0,Y 464.961,Z 269.815,A -85,B 0,C 180,E1 22518.298,E2 22518.298} C_VEL
LIN {X 0,Y 464.998,Z 269.804,A -85,B 0,C 180,E1 22514.698,E2 22514.698} C_VEL
LIN {X 0,Y 464.967,Z 269.804,A -85,B 0,C 180,E1 22511.033,E2 22511.033} C_VEL
LIN {X 0,Y 464.942,Z 269.808,A -85,B 0,C 180,E1 22507.538,E2 22507.538} C_VEL
LIN {X 0,Y 464.949,Z 269.811,A -85,B 0,C 180,E1 22503.811,E2 22503.811} C_VEL
LIN {X 0,Y 464.979,Z 269.813,A -85,B 0,C 180,E1 22500.246,E2 22500.246} C_VEL
LIN {X 0,Y 465.006,Z 269.814,A -85,B 0,C 180,E1 22496.619,E2 22496.619} C_VEL
LIN {X 0,Y 464.987,Z 269.806,A -85,B 0,C 180,E1 22492.959,E2 22492.959} C_VEL
LIN {X 0,Y 464.967,Z 269.801,A -85,B 0,C 180,E1 22489.343,E2 22489.343} C_VEL
LIN {X 0,Y 464.973,Z 269.803,A -85,B 0,C 180,E1 22485.682,E2 22485.682} C_VEL
LIN {X 0,Y 465.001,Z 269.802,A -85,B 0,C 180,E1 22482.092,E2 22482.092} C_VEL
LIN {X 0,Y 465.018,Z 269.803,A -85,B 0,C 180,E1 22478.427,E2 22478.427} C_VEL
LIN {X 0,Y 465.003,Z 269.808,A -85,B 0,C 180,E1 22474.802,E2 22474.802} C_VEL
LIN {X 0,Y 464.987,Z 269.811,A -85,B 0,C 180,E1 22471.206,E2 22471.206} C_VEL
LIN {X 0,Y 464.988,Z 269.787,A -85,B 0,C 180,E1 22467.446,E2 22467.446} C_VEL
LIN {X 0,Y 465.008,Z 269.787,A -85,B 0,C 180,E1 22463.903,E2 22463.903} C_VEL
LIN {X 0,Y 465.011,Z 269.814,A -85,B 0,C 180,E1 22460.312,E2 22460.312} C_VEL
LIN {X 0,Y 465.009,Z 269.785,A -85,B 0,C 180,E1 22456.614,E2 22456.614} C_VEL
LIN {X 0,Y 465.044,Z 270.042,A -85,B 0,C 180,E1 22453.897,E2 22453.897} C_VEL
LIN {X 0,Y 466.662,Z 273.807,A -85,B 0,C 180,E1 22453.241,E2 22453.241} C_VEL
LIN {X 0,Y 474.979,Z 292.554,A -85,B 0,C 180,E1 22450.356,E2 22450.356} C_VEL
LIN {X 0,Y 482.673,Z 311.789,A -85,B 0,C 180,E1 22447.701,E2 22447.701} C_VEL
LIN {X 0,Y 481.582,Z 327.093,A -85,B 0,C 180,E1 22446.419,E2 22446.419} C_VEL
LIN {X 0,Y 486.271,Z 354.665,A -85,B 0,C 180,E1 22445.484,E2 22445.484} C_VEL
LIN {X 0,Y 485.069,Z 425.29,A -85,B 0,C 180,E1 22444.37,E2 22444.37} C_VEL
LIN {X 0,Y 484.143,Z 432.989,A -85,B 0,C 180,E1 22444.321,E2 22444.321} C_VEL
LIN {X 0,Y 478.803,Z 453.526,A -85,B 0,C 180,E1 22444.448,E2 22444.448} C_VEL
LIN {X 0,Y 478.081,Z 460.135,A -85,B 0,C 180,E1 22444.399,E2 22444.399} C_VEL
LIN {X 0,Y 475.854,Z 593.567,A -85,B 0,C 180,E1 22442.282,E2 22442.282} C_VEL
LIN {X 0,Y 474.905,Z 613.805,A -85,B 0,C 180,E1 22441.747,E2 22441.747} C_VEL
LIN {X 0,Y 473.577,Z 633.56,A -85,B 0,C 180,E1 22441.007,E2 22441.007} C_VEL
LIN {X 0,Y 471.991,Z 652.639,A -85,B 0,C 180,E1 22440.065,E2 22440.065} C_VEL
LIN {X 0,Y 470.164,Z 670.931,A -85,B 0,C 180,E1 22438.933,E2 22438.933} C_VEL
LIN {X 0,Y 468.108,Z 689.017,A -85,B 0,C 180,E1 22437.55,E2 22437.55} C_VEL
LIN {X 0,Y 466.012,Z 705.431,A -85,B 0,C 180,E1 22436.024,E2 22436.024} C_VEL
LIN {X 0,Y 463.902,Z 721.365,A -85,B 0,C 180,E1 22434.258,E2 22434.258} C_VEL
LIN {X 0,Y 461.897,Z 736.511,A -85,B 0,C 180,E1 22432.26,E2 22432.26} C_VEL
LIN {X 0,Y 460.19,Z 749.821,A -85,B 0,C 180,E1 22430.18,E2 22430.18} C_VEL
LIN {X 0,Y 458.749,Z 762.139,A -85,B 0,C 180,E1 22427.897,E2 22427.897} C_VEL
LIN {X 0,Y 457.618,Z 773.091,A -85,B 0,C 180,E1 22425.459,E2 22425.459} C_VEL
LIN {X 0,Y 456.817,Z 782.461,A -85,B 0,C 180,E1 22422.9,E2 22422.9} C_VEL
LIN {X 0,Y 456.325,Z 789.969,A -85,B 0,C 180,E1 22420.323,E2 22420.323} C_VEL
LIN {X 0,Y 456.078,Z 795.577,A -85,B 0,C 180,E1 22417.812,E2 22417.812} C_VEL
LIN {X 0,Y 455.959,Z 799.788,A -85,B 0,C 180,E1 22415.158,E2 22415.158} C_VEL
LIN {X 0,Y 455.928,Z 802.211,A -85,B 0,C 180,E1 22412.64,E2 22412.64} C_VEL
LIN {X 0,Y 455.928,Z 803.101,A -85,B 0,C 180,E1 22410,E2 22410} C_VEL
LIN {X 0,Y 455.921,Z 802.325,A -85,B 0,C 180,E1 22407.486,E2 22407.486} C_VEL
LIN {X 0,Y 455.958,Z 800.052,A -85,B 0,C 180,E1 22404.968,E2 22404.968} C_VEL
LIN {X 0,Y 456.052,Z 796.241,A -85,B 0,C 180,E1 22402.441,E2 22402.441} C_VEL
LIN {X 0,Y 456.29,Z 790.811,A -85,B 0,C 180,E1 22399.904,E2 22399.904} C_VEL
LIN {X 0,Y 456.761,Z 783.182,A -85,B 0,C 180,E1 22397.227,E2 22397.227} C_VEL
LIN {X 0,Y 457.481,Z 774.429,A -85,B 0,C 180,E1 22394.796,E2 22394.796} C_VEL
LIN {X 0,Y 458.483,Z 764.378,A -85,B 0,C 180,E1 22392.486,E2 22392.486} C_VEL
LIN {X 0,Y 459.867,Z 752.363,A -85,B 0,C 180,E1 22390.174,E2 22390.174} C_VEL
LIN {X 0,Y 461.475,Z 739.752,A -85,B 0,C 180,E1 22388.121,E2 22388.121} C_VEL
LIN {X 0,Y 463.457,Z 724.852,A -85,B 0,C 180,E1 22386.073,E2 22386.073} C_VEL
LIN {X 0,Y 465.607,Z 708.763,A -85,B 0,C 180,E1 22384.225,E2 22384.225} C_VEL
LIN {X 0,Y 467.602,Z 692.901,A -85,B 0,C 180,E1 22382.7,E2 22382.7} C_VEL
LIN {X 0,Y 469.676,Z 675.309,A -85,B 0,C 180,E1 22381.292,E2 22381.292} C_VEL
LIN {X 0,Y 471.538,Z 657.395,A -85,B 0,C 180,E1 22380.113,E2 22380.113} C_VEL
LIN {X 0,Y 473.26,Z 638.328,A -85,B 0,C 180,E1 22379.111,E2 22379.111} C_VEL
LIN {X 0,Y 474.636,Z 618.248,A -85,B 0,C 180,E1 22378.308,E2 22378.308} C_VEL
LIN {X 0,Y 475.647,Z 598.3,A -85,B 0,C 180,E1 22377.738,E2 22377.738} C_VEL
LIN {X 0,Y 476.319,Z 571.307,A -85,B 0,C 180,E1 22377.25,E2 22377.25} C_VEL
LIN {X 0,Y 479.938,Z 354.912,A -85,B 0,C 180,E1 22373.832,E2 22373.832} C_VEL
LIN {X 0,Y 474.979,Z 326.025,A -85,B 0,C 180,E1 22372.796,E2 22372.796} C_VEL
LIN {X 0,Y 475.743,Z 314.896,A -85,B 0,C 180,E1 22371.816,E2 22371.816} C_VEL
LIN {X 0,Y 468.389,Z 296.461,A -85,B 0,C 180,E1 22369.217,E2 22369.217} C_VEL
LIN {X 0,Y 461.477,Z 280.97,A -85,B 0,C 180,E1 22366.793,E2 22366.793} C_VEL
LIN {X 0,Y 458.39,Z 274.3,A -85,B 0,C 180,E1 22365.68,E2 22365.68} C_VEL
LIN {X 0,Y 457.101,Z 271.018,A -85,B 0,C 180,E1 22365.084,E2 22365.084} C_VEL
LIN {X 0,Y 457.065,Z 270.769,A -85,B 0,C 180,E1 22361.517,E2 22361.517} C_VEL
LIN {X 0,Y 457.067,Z 270.766,A -85,B 0,C 180,E1 22357.844,E2 22357.844} C_VEL
LIN {X 0,Y 457.068,Z 270.801,A -85,B 0,C 180,E1 22354.208,E2 22354.208} C_VEL
LIN {X 0,Y 457.052,Z 270.764,A -85,B 0,C 180,E1 22350.47,E2 22350.47} C_VEL
LIN {X 0,Y 457.053,Z 270.794,A -85,B 0,C 180,E1 22346.786,E2 22346.786} C_VEL
LIN {X 0,Y 457.063,Z 270.792,A -85,B 0,C 180,E1 22343.053,E2 22343.053} C_VEL
LIN {X 0,Y 457.077,Z 270.793,A -85,B 0,C 180,E1 22339.421,E2 22339.421} C_VEL
LIN {X 0,Y 457.074,Z 270.8,A -85,B 0,C 180,E1 22335.739,E2 22335.739} C_VEL
LIN {X 0,Y 457.044,Z 270.802,A -85,B 0,C 180,E1 22332.08,E2 22332.08} C_VEL
LIN {X 0,Y 457.029,Z 270.803,A -85,B 0,C 180,E1 22328.429,E2 22328.429} C_VEL
LIN {X 0,Y 457.032,Z 270.802,A -85,B 0,C 180,E1 22324.769,E2 22324.769} C_VEL
LIN {X 0,Y 457.056,Z 270.791,A -85,B 0,C 180,E1 22321.128,E2 22321.128} C_VEL
LIN {X 0,Y 457.05,Z 270.793,A -85,B 0,C 180,E1 22317.618,E2 22317.618} C_VEL
LIN {X 0,Y 457.013,Z 270.805,A -85,B 0,C 180,E1 22314.098,E2 22314.098} C_VEL
LIN {X 0,Y 457.005,Z 270.806,A -85,B 0,C 180,E1 22310.429,E2 22310.429} C_VEL
LIN {X 0,Y 457.018,Z 270.806,A -85,B 0,C 180,E1 22306.79,E2 22306.79} C_VEL
LIN {X 0,Y 457.05,Z 270.797,A -85,B 0,C 180,E1 22303.216,E2 22303.216} C_VEL
LIN {X 0,Y 457.036,Z 270.798,A -85,B 0,C 180,E1 22299.511,E2 22299.511} C_VEL
LIN {X 0,Y 457.01,Z 270.802,A -85,B 0,C 180,E1 22295.988,E2 22295.988} C_VEL
LIN {X 0,Y 457.014,Z 270.806,A -85,B 0,C 180,E1 22292.225,E2 22292.225} C_VEL
LIN {X 0,Y 457.032,Z 270.763,A -85,B 0,C 180,E1 22288.623,E2 22288.623} C_VEL
LIN {X 0,Y 457.07,Z 270.793,A -85,B 0,C 180,E1 22285.031,E2 22285.031} C_VEL
LIN {X 0,Y 457.069,Z 270.794,A -85,B 0,C 180,E1 22281.271,E2 22281.271} C_VEL
LIN {X 0,Y 457.059,Z 270.996,A -85,B 0,C 180,E1 22277.952,E2 22277.952} C_VEL
LIN {X 0,Y 458.172,Z 273.972,A -85,B 0,C 180,E1 22277.429,E2 22277.429} C_VEL
LIN {X 0,Y 459.661,Z 276.861,A -85,B 0,C 180,E1 22276.958,E2 22276.958} C_VEL
LIN {X 0,Y 465.668,Z 289.281,A -85,B 0,C 180,E1 22275.057,E2 22275.057} C_VEL
LIN {X 0,Y 473.016,Z 305.268,A -85,B 0,C 180,E1 22272.843,E2 22272.843} C_VEL
LIN {X 0,Y 482.083,Z 320.762,A -85,B 0,C 180,E1 22271.626,E2 22271.626} C_VEL
LIN {X 0,Y 483.512,Z 331.045,A -85,B 0,C 180,E1 22271.29,E2 22271.29} C_VEL
LIN {X 0,Y 478.743,Z 543.234,A -85,B 0,C 180,E1 22267.694,E2 22267.694} C_VEL
LIN {X 0,Y 477.261,Z 608.711,A -85,B 0,C 180,E1 22266.571,E2 22266.571} C_VEL
LIN {X 0,Y 476.15,Z 630.339,A -85,B 0,C 180,E1 22265.998,E2 22265.998} C_VEL
LIN {X 0,Y 474.676,Z 652.576,A -85,B 0,C 180,E1 22265.187,E2 22265.187} C_VEL
LIN {X 0,Y 473.043,Z 673.383,A -85,B 0,C 180,E1 22264.21,E2 22264.21} C_VEL
LIN {X 0,Y 471.235,Z 693.382,A -85,B 0,C 180,E1 22263.044,E2 22263.044} C_VEL
LIN {X 0,Y 469.271,Z 712.701,A -85,B 0,C 180,E1 22261.681,E2 22261.681} C_VEL
LIN {X 0,Y 467.262,Z 731.396,A -85,B 0,C 180,E1 22260.117,E2 22260.117} C_VEL
LIN {X 0,Y 465.225,Z 749.281,A -85,B 0,C 180,E1 22258.357,E2 22258.357} C_VEL
LIN {X 0,Y 463.396,Z 765.116,A -85,B 0,C 180,E1 22256.527,E2 22256.527} C_VEL
LIN {X 0,Y 461.617,Z 780.795,A -85,B 0,C 180,E1 22254.437,E2 22254.437} C_VEL
LIN {X 0,Y 460.294,Z 792.593,A -85,B 0,C 180,E1 22252.603,E2 22252.603} C_VEL
LIN {X 0,Y 458.79,Z 806.259,A -85,B 0,C 180,E1 22250.067,E2 22250.067} C_VEL
LIN {X 0,Y 457.744,Z 817.23,A -85,B 0,C 180,E1 22247.675,E2 22247.675} C_VEL
LIN {X 0,Y 456.933,Z 827.052,A -85,B 0,C 180,E1 22245.093,E2 22245.093} C_VEL
LIN {X 0,Y 456.394,Z 835.469,A -85,B 0,C 180,E1 22242.397,E2 22242.397} C_VEL
LIN {X 0,Y 456.103,Z 842.129,A -85,B 0,C 180,E1 22239.718,E2 22239.718} C_VEL
LIN {X 0,Y 455.978,Z 846.813,A -85,B 0,C 180,E1 22237.18,E2 22237.18} C_VEL
LIN {X 0,Y 455.919,Z 850.331,A -85,B 0,C 180,E1 22234.402,E2 22234.402} C_VEL
LIN {X 0,Y 455.904,Z 852.085,A -85,B 0,C 180,E1 22231.885,E2 22231.885} C_VEL
LIN {X 0,Y 455.903,Z 852.371,A -85,B 0,C 180,E1 22229.246,E2 22229.246} C_VEL
LIN {X 0,Y 455.913,Z 851.235,A -85,B 0,C 180,E1 22226.605,E2 22226.605} C_VEL
LIN {X 0,Y 455.936,Z 848.616,A -85,B 0,C 180,E1 22224.084,E2 22224.084} C_VEL
LIN {X 0,Y 456.025,Z 844.415,A -85,B 0,C 180,E1 22221.426,E2 22221.426} C_VEL
LIN {X 0,Y 456.228,Z 838.856,A -85,B 0,C 180,E1 22218.881,E2 22218.881} C_VEL
LIN {X 0,Y 456.642,Z 831.286,A -85,B 0,C 180,E1 22216.193,E2 22216.193} C_VEL
LIN {X 0,Y 457.302,Z 822.379,A -85,B 0,C 180,E1 22213.618,E2 22213.618} C_VEL
LIN {X 0,Y 458.215,Z 812.091,A -85,B 0,C 180,E1 22211.159,E2 22211.159} C_VEL
LIN {X 0,Y 459.471,Z 799.858,A -85,B 0,C 180,E1 22208.691,E2 22208.691} C_VEL
LIN {X 0,Y 460.857,Z 787.737,A -85,B 0,C 180,E1 22206.595,E2 22206.595} C_VEL
LIN {X 0,Y 462.582,Z 772.293,A -85,B 0,C 180,E1 22204.388,E2 22204.388} C_VEL
LIN {X 0,Y 464.474,Z 755.75,A -85,B 0,C 180,E1 22202.362,E2 22202.362} C_VEL
LIN {X 0,Y 466.473,Z 738.286,A -85,B 0,C 180,E1 22200.527,E2 22200.527} C_VEL
LIN {X 0,Y 468.507,Z 720.129,A -85,B 0,C 180,E1 22198.906,E2 22198.906} C_VEL
LIN {X 0,Y 470.45,Z 701.125,A -85,B 0,C 180,E1 22197.473,E2 22197.473} C_VEL
LIN {X 0,Y 472.423,Z 680.457,A -85,B 0,C 180,E1 22196.178,E2 22196.178} C_VEL
LIN {X 0,Y 474.137,Z 660.3,A -85,B 0,C 180,E1 22195.147,E2 22195.147} C_VEL
LIN {X 0,Y 475.594,Z 638.949,A -85,B 0,C 180,E1 22194.288,E2 22194.288} C_VEL
LIN {X 0,Y 476.912,Z 616.011,A -85,B 0,C 180,E1 22193.605,E2 22193.605} C_VEL
LIN {X 0,Y 477.729,Z 593.56,A -85,B 0,C 180,E1 22193.146,E2 22193.146} C_VEL
LIN {X 0,Y 482.376,Z 380.021,A -85,B 0,C 180,E1 22189.547,E2 22189.547} C_VEL
LIN {X 0,Y 483.376,Z 328.84,A -85,B 0,C 180,E1 22188.654,E2 22188.654} C_VEL
LIN {X 0,Y 481.751,Z 319.827,A -85,B 0,C 180,E1 22188.323,E2 22188.323} C_VEL
LIN {X 0,Y 472.431,Z 304.183,A -85,B 0,C 180,E1 22187.042,E2 22187.042} C_VEL
LIN {X 0,Y 464.461,Z 286.617,A -85,B 0,C 180,E1 22184.559,E2 22184.559} C_VEL
LIN {X 0,Y 458.592,Z 274.594,A -85,B 0,C 180,E1 22182.692,E2 22182.692} C_VEL
LIN {X 0,Y 457.068,Z 271.041,A -85,B 0,C 180,E1 22182.074,E2 22182.074} C_VEL
LIN {X 0,Y 457.082,Z 270.8,A -85,B 0,C 180,E1 22179.049,E2 22179.049} C_VEL
LIN {X 0,Y 457.039,Z 270.784,A -85,B 0,C 180,E1 22175.432,E2 22175.432} C_VEL
LIN {X 0,Y 457.017,Z 270.767,A -85,B 0,C 180,E1 22171.82,E2 22171.82} C_VEL
LIN {X 0,Y 457.023,Z 270.807,A -85,B 0,C 180,E1 22168.159,E2 22168.159} C_VEL
LIN {X 0,Y 457.047,Z 270.803,A -85,B 0,C 180,E1 22164.56,E2 22164.56} C_VEL
LIN {X 0,Y 457.058,Z 270.802,A -85,B 0,C 180,E1 22160.92,E2 22160.92} C_VEL
LIN {X 0,Y 457.014,Z 270.806,A -85,B 0,C 180,E1 22157.31,E2 22157.31} C_VEL
LIN {X 0,Y 456.996,Z 270.807,A -85,B 0,C 180,E1 22153.737,E2 22153.737} C_VEL
LIN {X 0,Y 457.011,Z 270.806,A -85,B 0,C 180,E1 22150.08,E2 22150.08} C_VEL
LIN {X 0,Y 457.056,Z 270.793,A -85,B 0,C 180,E1 22146.532,E2 22146.532} C_VEL
LIN {X 0,Y 457.046,Z 270.791,A -85,B 0,C 180,E1 22142.884,E2 22142.884} C_VEL
LIN {X 0,Y 457.017,Z 270.802,A -85,B 0,C 180,E1 22139.373,E2 22139.373} C_VEL
LIN {X 0,Y 457.021,Z 270.804,A -85,B 0,C 180,E1 22135.734,E2 22135.734} C_VEL
LIN {X 0,Y 457.056,Z 270.802,A -85,B 0,C 180,E1 22132.205,E2 22132.205} C_VEL
LIN {X 0,Y 457.073,Z 270.795,A -85,B 0,C 180,E1 22128.517,E2 22128.517} C_VEL
LIN {X 0,Y 457.055,Z 270.791,A -85,B 0,C 180,E1 22124.91,E2 22124.91} C_VEL
LIN {X 0,Y 457.04,Z 270.791,A -85,B 0,C 180,E1 22121.241,E2 22121.241} C_VEL
LIN {X 0,Y 457.042,Z 270.791,A -85,B 0,C 180,E1 22117.49,E2 22117.49} C_VEL
LIN {X 0,Y 457.056,Z 270.79,A -85,B 0,C 180,E1 22113.775,E2 22113.775} C_VEL
LIN {X 0,Y 457.075,Z 270.776,A -85,B 0,C 180,E1 22110.227,E2 22110.227} C_VEL
LIN {X 0,Y 457.073,Z 270.793,A -85,B 0,C 180,E1 22106.452,E2 22106.452} C_VEL
LIN {X 0,Y 457.066,Z 270.762,A -85,B 0,C 180,E1 22102.702,E2 22102.702} C_VEL
LIN {X 0,Y 457.062,Z 270.78,A -85,B 0,C 180,E1 22098.999,E2 22098.999} C_VEL
LIN {X 0,Y 457.063,Z 270.8,A -85,B 0,C 180,E1 22095.219,E2 22095.219} C_VEL
LIN {X 0,Y 457.143,Z 271.262,A -85,B 0,C 180,E1 22094.743,E2 22094.743} C_VEL
LIN {X 0,Y 464.599,Z 287.812,A -85,B 0,C 180,E1 22092.012,E2 22092.012} C_VEL
LIN {X 0,Y 471.82,Z 304.836,A -85,B 0,C 180,E1 22089.474,E2 22089.474} C_VEL
LIN {X 0,Y 475.831,Z 315.754,A -85,B 0,C 180,E1 22088,E2 22088} C_VEL
LIN {X 0,Y 475.048,Z 327.008,A -85,B 0,C 180,E1 22087.061,E2 22087.061} C_VEL
LIN {X 0,Y 479.957,Z 355.994,A -85,B 0,C 180,E1 22086.053,E2 22086.053} C_VEL
LIN {X 0,Y 478.081,Z 460.135,A -85,B 0,C 180,E1 22084.399,E2 22084.399} C_VEL
LIN {X 0,Y 477.152,Z 467.834,A -85,B 0,C 180,E1 22084.351,E2 22084.351} C_VEL
LIN {X 0,Y 471.836,Z 488.374,A -85,B 0,C 180,E1 22084.48,E2 22084.48} C_VEL
LIN {X 0,Y 471.107,Z 494.983,A -85,B 0,C 180,E1 22084.432,E2 22084.432} C_VEL
LIN {X 0,Y 469.32,Z 593.852,A -85,B 0,C 180,E1 22082.841,E2 22082.841} C_VEL
LIN {X 0,Y 468.328,Z 614.04,A -85,B 0,C 180,E1 22082.303,E2 22082.303} C_VEL
LIN {X 0,Y 466.936,Z 633.683,A -85,B 0,C 180,E1 22081.563,E2 22081.563} C_VEL
LIN {X 0,Y 465.164,Z 653.851,A -85,B 0,C 180,E1 22080.553,E2 22080.553} C_VEL
LIN {X 0,Y 463.237,Z 672.01,A -85,B 0,C 180,E1 22079.408,E2 22079.408} C_VEL
LIN {X 0,Y 461.069,Z 690.156,A -85,B 0,C 180,E1 22078.001,E2 22078.001} C_VEL
LIN {X 0,Y 458.797,Z 707.16,A -85,B 0,C 180,E1 22076.396,E2 22076.396} C_VEL
LIN {X 0,Y 456.665,Z 722.329,A -85,B 0,C 180,E1 22074.682,E2 22074.682} C_VEL
LIN {X 0,Y 454.624,Z 736.615,A -85,B 0,C 180,E1 22072.772,E2 22072.772} C_VEL
LIN {X 0,Y 452.782,Z 749.806,A -85,B 0,C 180,E1 22070.69,E2 22070.69} C_VEL
LIN {X 0,Y 451.163,Z 762.305,A -85,B 0,C 180,E1 22068.342,E2 22068.342} C_VEL
LIN {X 0,Y 449.854,Z 773.659,A -85,B 0,C 180,E1 22065.761,E2 22065.761} C_VEL
LIN {X 0,Y 448.957,Z 783.073,A -85,B 0,C 180,E1 22063.13,E2 22063.13} C_VEL
LIN {X 0,Y 448.4,Z 790.631,A -85,B 0,C 180,E1 22060.466,E2 22060.466} C_VEL
LIN {X 0,Y 448.122,Z 796.088,A -85,B 0,C 180,E1 22057.951,E2 22057.951} C_VEL
LIN {X 0,Y 447.981,Z 800.26,A -85,B 0,C 180,E1 22055.25,E2 22055.25} C_VEL
LIN {X 0,Y 447.943,Z 802.665,A -85,B 0,C 180,E1 22052.687,E2 22052.687} C_VEL
LIN {X 0,Y 447.941,Z 803.55,A -85,B 0,C 180,E1 22050,E2 22050} C_VEL
LIN {X 0,Y 447.935,Z 802.777,A -85,B 0,C 180,E1 22047.441,E2 22047.441} C_VEL
LIN {X 0,Y 447.979,Z 800.522,A -85,B 0,C 180,E1 22044.878,E2 22044.878} C_VEL
LIN {X 0,Y 448.092,Z 796.743,A -85,B 0,C 180,E1 22042.306,E2 22042.306} C_VEL
LIN {X 0,Y 448.364,Z 791.353,A -85,B 0,C 180,E1 22039.724,E2 22039.724} C_VEL
LIN {X 0,Y 448.858,Z 784.157,A -85,B 0,C 180,E1 22037.129,E2 22037.129} C_VEL
LIN {X 0,Y 449.64,Z 775.576,A -85,B 0,C 180,E1 22034.656,E2 22034.656} C_VEL
LIN {X 0,Y 450.799,Z 765.126,A -85,B 0,C 180,E1 22032.177,E2 22032.177} C_VEL
LIN {X 0,Y 452.312,Z 753.222,A -85,B 0,C 180,E1 22029.828,E2 22029.828} C_VEL
LIN {X 0,Y 454.053,Z 740.725,A -85,B 0,C 180,E1 22027.744,E2 22027.744} C_VEL
LIN {X 0,Y 456.174,Z 725.913,A -85,B 0,C 180,E1 22025.666,E2 22025.666} C_VEL
LIN {X 0,Y 458.359,Z 710.389,A -85,B 0,C 180,E1 22023.856,E2 22023.856} C_VEL
LIN {X 0,Y 460.516,Z 694.183,A -85,B 0,C 180,E1 22022.269,E2 22022.269} C_VEL
LIN {X 0,Y 462.803,Z 675.768,A -85,B 0,C 180,E1 22020.775,E2 22020.775} C_VEL
LIN {X 0,Y 464.823,Z 657.281,A -85,B 0,C 180,E1 22019.552,E2 22019.552} C_VEL
LIN {X 0,Y 466.615,Z 638.31,A -85,B 0,C 180,E1 22018.55,E2 22018.55} C_VEL
LIN {X 0,Y 468.09,Z 617.895,A -85,B 0,C 180,E1 22017.731,E2 22017.731} C_VEL
LIN {X 0,Y 469.132,Z 598.045,A -85,B 0,C 180,E1 22017.167,E2 22017.167} C_VEL
LIN {X 0,Y 469.836,Z 570.526,A -85,B 0,C 180,E1 22016.67,E2 22016.67} C_VEL
LIN {X 0,Y 473.66,Z 356.21,A -85,B 0,C 180,E1 22013.245,E2 22013.245} C_VEL
LIN {X 0,Y 468.481,Z 325.568,A -85,B 0,C 180,E1 22012.112,E2 22012.112} C_VEL
LIN {X 0,Y 469.017,Z 318.482,A -85,B 0,C 180,E1 22011.479,E2 22011.479} C_VEL
LIN {X 0,Y 461.673,Z 300.034,A -85,B 0,C 180,E1 22008.825,E2 22008.825} C_VEL
LIN {X 0,Y 454.427,Z 283.594,A -85,B 0,C 180,E1 22006.194,E2 22006.194} C_VEL
LIN {X 0,Y 450.394,Z 275.21,A -85,B 0,C 180,E1 22004.727,E2 22004.727} C_VEL
LIN {X 0,Y 449.16,Z 271.977,A -85,B 0,C 180,E1 22004.125,E2 22004.125} C_VEL
LIN {X 0,Y 449.125,Z 271.776,A -85,B 0,C 180,E1 22000.546,E2 22000.546} C_VEL
LIN {X 0,Y 449.118,Z 271.752,A -85,B 0,C 180,E1 21996.733,E2 21996.733} C_VEL
LIN {X 0,Y 449.126,Z 271.773,A -85,B 0,C 180,E1 21993.054,E2 21993.054} C_VEL
LIN {X 0,Y 449.136,Z 271.771,A -85,B 0,C 180,E1 21989.325,E2 21989.325} C_VEL
LIN {X 0,Y 449.136,Z 271.778,A -85,B 0,C 180,E1 21985.587,E2 21985.587} C_VEL
LIN {X 0,Y 449.138,Z 271.777,A -85,B 0,C 180,E1 21981.825,E2 21981.825} C_VEL
LIN {X 0,Y 449.115,Z 271.78,A -85,B 0,C 180,E1 21978.085,E2 21978.085} C_VEL
LIN {X 0,Y 449.098,Z 271.778,A -85,B 0,C 180,E1 21974.432,E2 21974.432} C_VEL
LIN {X 0,Y 449.096,Z 271.777,A -85,B 0,C 180,E1 21970.649,E2 21970.649} C_VEL
LIN {X 0,Y 449.113,Z 271.783,A -85,B 0,C 180,E1 21967.034,E2 21967.034} C_VEL
LIN {X 0,Y 449.129,Z 271.791,A -85,B 0,C 180,E1 21963.318,E2 21963.318} C_VEL
LIN {X 0,Y 449.116,Z 271.79,A -85,B 0,C 180,E1 21959.618,E2 21959.618} C_VEL
LIN {X 0,Y 449.079,Z 271.789,A -85,B 0,C 180,E1 21956.043,E2 21956.043} C_VEL
LIN {X 0,Y 449.068,Z 271.785,A -85,B 0,C 180,E1 21952.323,E2 21952.323} C_VEL
LIN {X 0,Y 449.075,Z 271.781,A -85,B 0,C 180,E1 21948.701,E2 21948.701} C_VEL
LIN {X 0,Y 449.102,Z 271.78,A -85,B 0,C 180,E1 21945.063,E2 21945.063} C_VEL
LIN {X 0,Y 449.11,Z 271.782,A -85,B 0,C 180,E1 21941.302,E2 21941.302} C_VEL
LIN {X 0,Y 449.077,Z 271.791,A -85,B 0,C 180,E1 21937.759,E2 21937.759} C_VEL
LIN {X 0,Y 449.074,Z 271.79,A -85,B 0,C 180,E1 21934.089,E2 21934.089} C_VEL
LIN {X 0,Y 449.081,Z 271.775,A -85,B 0,C 180,E1 21930.378,E2 21930.378} C_VEL
LIN {X 0,Y 449.114,Z 271.778,A -85,B 0,C 180,E1 21926.793,E2 21926.793} C_VEL
LIN {X 0,Y 449.124,Z 271.751,A -85,B 0,C 180,E1 21923.212,E2 21923.212} C_VEL
LIN {X 0,Y 449.1,Z 271.767,A -85,B 0,C 180,E1 21919.619,E2 21919.619} C_VEL
LIN {X 0,Y 449.202,Z 272.214,A -85,B 0,C 180,E1 21918.829,E2 21918.829} C_VEL
LIN {X 0,Y 450.614,Z 275.554,A -85,B 0,C 180,E1 21918.267,E2 21918.267} C_VEL
LIN {X 0,Y 455.777,Z 285.992,A -85,B 0,C 180,E1 21916.561,E2 21916.561} C_VEL
LIN {X 0,Y 463.691,Z 302.956,A -85,B 0,C 180,E1 21914.018,E2 21914.018} C_VEL
LIN {X 0,Y 465.234,Z 306.143,A -85,B 0,C 180,E1 21913.637,E2 21913.637} C_VEL
LIN {X 0,Y 476.215,Z 324.621,A -85,B 0,C 180,E1 21912.126,E2 21912.126} C_VEL
LIN {X 0,Y 477.243,Z 332.561,A -85,B 0,C 180,E1 21911.866,E2 21911.866} C_VEL
LIN {X 0,Y 471.927,Z 549.518,A -85,B 0,C 180,E1 21908.122,E2 21908.122} C_VEL
LIN {X 0,Y 470.475,Z 608.455,A -85,B 0,C 180,E1 21907.091,E2 21907.091} C_VEL
LIN {X 0,Y 469.285,Z 630.274,A -85,B 0,C 180,E1 21906.503,E2 21906.503} C_VEL
LIN {X 0,Y 467.76,Z 651.984,A -85,B 0,C 180,E1 21905.699,E2 21905.699} C_VEL
LIN {X 0,Y 466.035,Z 672.628,A -85,B 0,C 180,E1 21904.723,E2 21904.723} C_VEL
LIN {X 0,Y 464.132,Z 692.653,A -85,B 0,C 180,E1 21903.542,E2 21903.542} C_VEL
LIN {X 0,Y 462.051,Z 712.06,A -85,B 0,C 180,E1 21902.162,E2 21902.162} C_VEL
LIN {X 0,Y 459.933,Z 730.909,A -85,B 0,C 180,E1 21900.576,E2 21900.576} C_VEL
LIN {X 0,Y 457.884,Z 747.988,A -85,B 0,C 180,E1 21898.879,E2 21898.879} C_VEL
LIN {X 0,Y 455.87,Z 764.478,A -85,B 0,C 180,E1 21896.96,E2 21896.96} C_VEL
LIN {X 0,Y 453.984,Z 780.091,A -85,B 0,C 180,E1 21894.853,E2 21894.853} C_VEL
LIN {X 0,Y 452.338,Z 794.243,A -85,B 0,C 180,E1 21892.619,E2 21892.619} C_VEL
LIN {X 0,Y 450.943,Z 807.093,A -85,B 0,C 180,E1 21890.236,E2 21890.236} C_VEL
LIN {X 0,Y 449.913,Z 817.275,A -85,B 0,C 180,E1 21887.981,E2 21887.981} C_VEL
LIN {X 0,Y 449.034,Z 827.051,A -85,B 0,C 180,E1 21885.365,E2 21885.365} C_VEL
LIN {X 0,Y 448.446,Z 835.468,A -85,B 0,C 180,E1 21882.621,E2 21882.621} C_VEL
LIN {X 0,Y 448.121,Z 842.129,A -85,B 0,C 180,E1 21879.892,E2 21879.892} C_VEL
LIN {X 0,Y 447.98,Z 846.812,A -85,B 0,C 180,E1 21877.309,E2 21877.309} C_VEL
LIN {X 0,Y 447.92,Z 850.331,A -85,B 0,C 180,E1 21874.481,E2 21874.481} C_VEL
LIN {X 0,Y 447.905,Z 852.085,A -85,B 0,C 180,E1 21871.919,E2 21871.919} C_VEL
LIN {X 0,Y 447.904,Z 852.371,A -85,B 0,C 180,E1 21869.233,E2 21869.233} C_VEL
LIN {X 0,Y 447.912,Z 851.235,A -85,B 0,C 180,E1 21866.545,E2 21866.545} C_VEL
LIN {X 0,Y 447.94,Z 848.616,A -85,B 0,C 180,E1 21863.978,E2 21863.978} C_VEL
LIN {X 0,Y 448.033,Z 844.415,A -85,B 0,C 180,E1 21861.272,E2 21861.272} C_VEL
LIN {X 0,Y 448.262,Z 838.856,A -85,B 0,C 180,E1 21858.68,E2 21858.68} C_VEL
LIN {X 0,Y 448.718,Z 831.285,A -85,B 0,C 180,E1 21855.944,E2 21855.944} C_VEL
LIN {X 0,Y 449.436,Z 822.378,A -85,B 0,C 180,E1 21853.323,E2 21853.323} C_VEL
LIN {X 0,Y 450.434,Z 812.09,A -85,B 0,C 180,E1 21850.821,E2 21850.821} C_VEL
LIN {X 0,Y 451.67,Z 800.2,A -85,B 0,C 180,E1 21848.441,E2 21848.441} C_VEL
LIN {X 0,Y 453.179,Z 786.995,A -85,B 0,C 180,E1 21846.187,E2 21846.187} C_VEL
LIN {X 0,Y 455.035,Z 771.397,A -85,B 0,C 180,E1 21843.931,E2 21843.931} C_VEL
LIN {X 0,Y 457.064,Z 754.743,A -85,B 0,C 180,E1 21841.874,E2 21841.874} C_VEL
LIN {X 0,Y 459.171,Z 737.211,A -85,B 0,C 180,E1 21840.018,E2 21840.018} C_VEL
LIN {X 0,Y 461.342,Z 718.787,A -85,B 0,C 180,E1 21838.368,E2 21838.368} C_VEL
LIN {X 0,Y 463.393,Z 699.482,A -85,B 0,C 180,E1 21836.915,E2 21836.915} C_VEL
LIN {X 0,Y 465.498,Z 678.519,A -85,B 0,C 180,E1 21835.605,E2 21835.605} C_VEL
LIN {X 0,Y 467.306,Z 658.122,A -85,B 0,C 180,E1 21834.562,E2 21834.562} C_VEL
LIN {X 0,Y 468.897,Z 636.18,A -85,B 0,C 180,E1 21833.691,E2 21833.691} C_VEL
LIN {X 0,Y 470.179,Z 614.533,A -85,B 0,C 180,E1 21833.058,E2 21833.058} C_VEL
LIN {X 0,Y 471.031,Z 590.734,A -85,B 0,C 180,E1 21832.578,E2 21832.578} C_VEL
LIN {X 0,Y 476.355,Z 368.201,A -85,B 0,C 180,E1 21828.75,E2 21828.75} C_VEL
LIN {X 0,Y 477.126,Z 330.371,A -85,B 0,C 180,E1 21828.078,E2 21828.078} C_VEL
LIN {X 0,Y 475.898,Z 323.816,A -85,B 0,C 180,E1 21827.827,E2 21827.827} C_VEL
LIN {X 0,Y 464.487,Z 304.848,A -85,B 0,C 180,E1 21826.236,E2 21826.236} C_VEL
LIN {X 0,Y 456.779,Z 288.02,A -85,B 0,C 180,E1 21823.765,E2 21823.765} C_VEL
LIN {X 0,Y 451.036,Z 276.13,A -85,B 0,C 180,E1 21821.855,E2 21821.855} C_VEL
LIN {X 0,Y 449.244,Z 272.446,A -85,B 0,C 180,E1 21821.215,E2 21821.215} C_VEL
LIN {X 0,Y 449.144,Z 271.811,A -85,B 0,C 180,E1 21820.88,E2 21820.88} C_VEL
LIN {X 0,Y 449.123,Z 271.752,A -85,B 0,C 180,E1 21817.158,E2 21817.158} C_VEL
LIN {X 0,Y 449.093,Z 271.789,A -85,B 0,C 180,E1 21813.514,E2 21813.514} C_VEL
LIN {X 0,Y 449.076,Z 271.768,A -85,B 0,C 180,E1 21809.916,E2 21809.916} C_VEL
LIN {X 0,Y 449.087,Z 271.786,A -85,B 0,C 180,E1 21806.299,E2 21806.299} C_VEL
LIN {X 0,Y 449.116,Z 271.782,A -85,B 0,C 180,E1 21802.653,E2 21802.653} C_VEL
LIN {X 0,Y 449.105,Z 271.78,A -85,B 0,C 180,E1 21798.968,E2 21798.968} C_VEL
LIN {X 0,Y 449.066,Z 271.782,A -85,B 0,C 180,E1 21795.364,E2 21795.364} C_VEL
LIN {X 0,Y 449.057,Z 271.783,A -85,B 0,C 180,E1 21791.69,E2 21791.69} C_VEL
LIN {X 0,Y 449.073,Z 271.786,A -85,B 0,C 180,E1 21788.063,E2 21788.063} C_VEL
LIN {X 0,Y 449.113,Z 271.789,A -85,B 0,C 180,E1 21784.469,E2 21784.469} C_VEL
LIN {X 0,Y 449.135,Z 271.791,A -85,B 0,C 180,E1 21780.638,E2 21780.638} C_VEL
LIN {X 0,Y 449.107,Z 271.789,A -85,B 0,C 180,E1 21776.937,E2 21776.937} C_VEL
LIN {X 0,Y 449.085,Z 271.783,A -85,B 0,C 180,E1 21773.351,E2 21773.351} C_VEL
LIN {X 0,Y 449.088,Z 271.777,A -85,B 0,C 180,E1 21769.61,E2 21769.61} C_VEL
LIN {X 0,Y 449.107,Z 271.779,A -85,B 0,C 180,E1 21765.956,E2 21765.956} C_VEL
LIN {X 0,Y 449.136,Z 271.78,A -85,B 0,C 180,E1 21762.322,E2 21762.322} C_VEL
LIN {X 0,Y 449.139,Z 271.781,A -85,B 0,C 180,E1 21758.515,E2 21758.515} C_VEL
LIN {X 0,Y 449.123,Z 271.786,A -85,B 0,C 180,E1 21754.836,E2 21754.836} C_VEL
LIN {X 0,Y 449.113,Z 271.784,A -85,B 0,C 180,E1 21751.111,E2 21751.111} C_VEL
LIN {X 0,Y 449.11,Z 271.761,A -85,B 0,C 180,E1 21747.4,E2 21747.4} C_VEL
LIN {X 0,Y 449.122,Z 271.757,A -85,B 0,C 180,E1 21743.688,E2 21743.688} C_VEL
LIN {X 0,Y 449.137,Z 271.79,A -85,B 0,C 180,E1 21739.956,E2 21739.956} C_VEL
LIN {X 0,Y 449.129,Z 271.77,A -85,B 0,C 180,E1 21736.16,E2 21736.16} C_VEL
LIN {X 0,Y 449.204,Z 272.248,A -85,B 0,C 180,E1 21735.698,E2 21735.698} C_VEL
LIN {X 0,Y 450.908,Z 275.95,A -85,B 0,C 180,E1 21735.019,E2 21735.019} C_VEL
LIN {X 0,Y 458.288,Z 292.171,A -85,B 0,C 180,E1 21732.302,E2 21732.302} C_VEL
LIN {X 0,Y 465.424,Z 309.18,A -85,B 0,C 180,E1 21729.728,E2 21729.728} C_VEL
LIN {X 0,Y 469.069,Z 318.93,A -85,B 0,C 180,E1 21728.378,E2 21728.378} C_VEL
LIN {X 0,Y 468.539,Z 326.733,A -85,B 0,C 180,E1 21727.729,E2 21727.729} C_VEL
LIN {X 0,Y 473.69,Z 357.38,A -85,B 0,C 180,E1 21726.636,E2 21726.636} C_VEL
LIN {X 0,Y 471.107,Z 494.983,A -85,B 0,C 180,E1 21724.432,E2 21724.432} C_VEL
LIN {X 0,Y 470.163,Z 502.683,A -85,B 0,C 180,E1 21724.385,E2 21724.385} C_VEL
LIN {X 0,Y 464.834,Z 523.221,A -85,B 0,C 180,E1 21724.518,E2 21724.518} C_VEL
LIN {X 0,Y 464.109,Z 529.829,A -85,B 0,C 180,E1 21724.469,E2 21724.469} C_VEL
LIN {X 0,Y 462.801,Z 594.536,A -85,B 0,C 180,E1 21723.406,E2 21723.406} C_VEL
LIN {X 0,Y 461.753,Z 614.736,A -85,B 0,C 180,E1 21722.858,E2 21722.858} C_VEL
LIN {X 0,Y 460.291,Z 634.21,A -85,B 0,C 180,E1 21722.113,E2 21722.113} C_VEL
LIN {X 0,Y 458.477,Z 653.844,A -85,B 0,C 180,E1 21721.121,E2 21721.121} C_VEL
LIN {X 0,Y 456.444,Z 672.099,A -85,B 0,C 180,E1 21719.962,E2 21719.962} C_VEL
LIN {X 0,Y 454.141,Z 690.323,A -85,B 0,C 180,E1 21718.538,E2 21718.538} C_VEL
LIN {X 0,Y 451.736,Z 707.393,A -85,B 0,C 180,E1 21716.912,E2 21716.912} C_VEL
LIN {X 0,Y 449.439,Z 722.893,A -85,B 0,C 180,E1 21715.144,E2 21715.144} C_VEL
LIN {X 0,Y 447.232,Z 737.488,A -85,B 0,C 180,E1 21713.17,E2 21713.17} C_VEL
LIN {X 0,Y 445.27,Z 750.666,A -85,B 0,C 180,E1 21711.055,E2 21711.055} C_VEL
LIN {X 0,Y 443.606,Z 762.49,A -85,B 0,C 180,E1 21708.799,E2 21708.799} C_VEL
LIN {X 0,Y 442.196,Z 773.414,A -85,B 0,C 180,E1 21706.282,E2 21706.282} C_VEL
LIN {X 0,Y 441.214,Z 782.399,A -85,B 0,C 180,E1 21703.765,E2 21703.765} C_VEL
LIN {X 0,Y 440.559,Z 789.999,A -85,B 0,C 180,E1 21701.122,E2 21701.122} C_VEL
LIN {X 0,Y 440.193,Z 796.109,A -85,B 0,C 180,E1 21698.358,E2 21698.358} C_VEL
LIN {X 0,Y 440.02,Z 800.278,A -85,B 0,C 180,E1 21695.738,E2 21695.738} C_VEL
LIN {X 0,Y 439.962,Z 802.98,A -85,B 0,C 180,E1 21692.996,E2 21692.996} C_VEL
LIN {X 0,Y 439.947,Z 803.955,A -85,B 0,C 180,E1 21690.26,E2 21690.26} C_VEL
LIN {X 0,Y 439.95,Z 803.36,A -85,B 0,C 180,E1 21687.656,E2 21687.656} C_VEL
LIN {X 0,Y 439.999,Z 801.146,A -85,B 0,C 180,E1 21684.916,E2 21684.916} C_VEL
LIN {X 0,Y 440.125,Z 797.49,A -85,B 0,C 180,E1 21682.297,E2 21682.297} C_VEL
LIN {X 0,Y 440.441,Z 791.893,A -85,B 0,C 180,E1 21679.537,E2 21679.537} C_VEL
LIN {X 0,Y 440.999,Z 784.755,A -85,B 0,C 180,E1 21676.896,E2 21676.896} C_VEL
LIN {X 0,Y 441.861,Z 776.252,A -85,B 0,C 180,E1 21674.379,E2 21674.379} C_VEL
LIN {X 0,Y 443.131,Z 765.893,A -85,B 0,C 180,E1 21671.858,E2 21671.858} C_VEL
LIN {X 0,Y 444.773,Z 754.085,A -85,B 0,C 180,E1 21669.471,E2 21669.471} C_VEL
LIN {X 0,Y 446.638,Z 741.614,A -85,B 0,C 180,E1 21667.354,E2 21667.354} C_VEL
LIN {X 0,Y 448.875,Z 726.74,A -85,B 0,C 180,E1 21665.244,E2 21665.244} C_VEL
LIN {X 0,Y 451.183,Z 711.224,A -85,B 0,C 180,E1 21663.408,E2 21663.408} C_VEL
LIN {X 0,Y 453.497,Z 694.855,A -85,B 0,C 180,E1 21661.781,E2 21661.781} C_VEL
LIN {X 0,Y 455.876,Z 676.729,A -85,B 0,C 180,E1 21660.286,E2 21660.286} C_VEL
LIN {X 0,Y 457.976,Z 658.697,A -85,B 0,C 180,E1 21659.068,E2 21659.068} C_VEL
LIN {X 0,Y 459.886,Z 639.525,A -85,B 0,C 180,E1 21658.036,E2 21658.036} C_VEL
LIN {X 0,Y 461.413,Z 619.644,A -85,B 0,C 180,E1 21657.217,E2 21657.217} C_VEL
LIN {X 0,Y 462.568,Z 599.483,A -85,B 0,C 180,E1 21656.622,E2 21656.622} C_VEL
LIN {X 0,Y 463.315,Z 573.855,A -85,B 0,C 180,E1 21656.14,E2 21656.14} C_VEL
LIN {X 0,Y 467.464,Z 357.731,A -85,B 0,C 180,E1 21652.65,E2 21652.65} C_VEL
LIN {X 0,Y 462.035,Z 325.651,A -85,B 0,C 180,E1 21651.448,E2 21651.448} C_VEL
LIN {X 0,Y 462.315,Z 322.056,A -85,B 0,C 180,E1 21651.131,E2 21651.131} C_VEL
LIN {X 0,Y 454.856,Z 303.221,A -85,B 0,C 180,E1 21648.365,E2 21648.365} C_VEL
LIN {X 0,Y 447.017,Z 285.408,A -85,B 0,C 180,E1 21645.431,E2 21645.431} C_VEL
LIN {X 0,Y 442.481,Z 276.227,A -85,B 0,C 180,E1 21643.746,E2 21643.746} C_VEL
LIN {X 0,Y 441.215,Z 272.931,A -85,B 0,C 180,E1 21643.099,E2 21643.099} C_VEL
LIN {X 0,Y 441.197,Z 272.774,A -85,B 0,C 180,E1 21639.387,E2 21639.387} C_VEL
LIN {X 0,Y 441.19,Z 272.758,A -85,B 0,C 180,E1 21635.554,E2 21635.554} C_VEL
LIN {X 0,Y 441.193,Z 272.733,A -85,B 0,C 180,E1 21631.808,E2 21631.808} C_VEL
LIN {X 0,Y 441.199,Z 272.778,A -85,B 0,C 180,E1 21627.977,E2 21627.977} C_VEL
LIN {X 0,Y 441.179,Z 272.78,A -85,B 0,C 180,E1 21624.218,E2 21624.218} C_VEL
LIN {X 0,Y 441.167,Z 272.781,A -85,B 0,C 180,E1 21620.567,E2 21620.567} C_VEL
LIN {X 0,Y 441.171,Z 272.783,A -85,B 0,C 180,E1 21616.864,E2 21616.864} C_VEL
LIN {X 0,Y 441.192,Z 272.772,A -85,B 0,C 180,E1 21613.232,E2 21613.232} C_VEL
LIN {X 0,Y 441.196,Z 272.765,A -85,B 0,C 180,E1 21609.391,E2 21609.391} C_VEL
LIN {X 0,Y 441.178,Z 272.764,A -85,B 0,C 180,E1 21605.723,E2 21605.723} C_VEL
LIN {X 0,Y 441.15,Z 272.772,A -85,B 0,C 180,E1 21602.078,E2 21602.078} C_VEL
LIN {X 0,Y 441.139,Z 272.78,A -85,B 0,C 180,E1 21598.442,E2 21598.442} C_VEL
LIN {X 0,Y 441.149,Z 272.784,A -85,B 0,C 180,E1 21594.799,E2 21594.799} C_VEL
LIN {X 0,Y 441.172,Z 272.779,A -85,B 0,C 180,E1 21591.135,E2 21591.135} C_VEL
LIN {X 0,Y 441.174,Z 272.773,A -85,B 0,C 180,E1 21587.301,E2 21587.301} C_VEL
LIN {X 0,Y 441.139,Z 272.772,A -85,B 0,C 180,E1 21583.677,E2 21583.677} C_VEL
LIN {X 0,Y 441.125,Z 272.774,A -85,B 0,C 180,E1 21580.124,E2 21580.124} C_VEL
LIN {X 0,Y 441.13,Z 272.777,A -85,B 0,C 180,E1 21576.301,E2 21576.301} C_VEL
LIN {X 0,Y 441.151,Z 272.779,A -85,B 0,C 180,E1 21572.607,E2 21572.607} C_VEL
LIN {X 0,Y 441.181,Z 272.734,A -85,B 0,C 180,E1 21568.942,E2 21568.942} C_VEL
LIN {X 0,Y 441.194,Z 272.769,A -85,B 0,C 180,E1 21565.121,E2 21565.121} C_VEL
LIN {X 0,Y 441.189,Z 272.766,A -85,B 0,C 180,E1 21561.282,E2 21561.282} C_VEL
LIN {X 0,Y 441.198,Z 273.087,A -85,B 0,C 180,E1 21559.886,E2 21559.886} C_VEL
LIN {X 0,Y 442.72,Z 276.552,A -85,B 0,C 180,E1 21559.256,E2 21559.256} C_VEL
LIN {X 0,Y 449.55,Z 290.207,A -85,B 0,C 180,E1 21556.937,E2 21556.937} C_VEL
LIN {X 0,Y 456.861,Z 305.879,A -85,B 0,C 180,E1 21554.572,E2 21554.572} C_VEL
LIN {X 0,Y 469.673,Z 327.031,A -85,B 0,C 180,E1 21552.74,E2 21552.74} C_VEL
LIN {X 0,Y 470.494,Z 329.15,A -85,B 0,C 180,E1 21552.612,E2 21552.612} C_VEL
LIN {X 0,Y 471.022,Z 334.247,A -85,B 0,C 180,E1 21552.455,E2 21552.455} C_VEL
LIN {X 0,Y 465.369,Z 549.584,A -85,B 0,C 180,E1 21548.685,E2 21548.685} C_VEL
LIN {X 0,Y 463.776,Z 608.063,A -85,B 0,C 180,E1 21547.636,E2 21547.636} C_VEL
LIN {X 0,Y 462.496,Z 629.849,A -85,B 0,C 180,E1 21547.037,E2 21547.037} C_VEL
LIN {X 0,Y 460.831,Z 652.011,A -85,B 0,C 180,E1 21546.201,E2 21546.201} C_VEL
LIN {X 0,Y 458.953,Z 673.052,A -85,B 0,C 180,E1 21545.185,E2 21545.185} C_VEL
LIN {X 0,Y 456.927,Z 693.277,A -85,B 0,C 180,E1 21543.97,E2 21543.97} C_VEL
LIN {X 0,Y 454.692,Z 712.849,A -85,B 0,C 180,E1 21542.543,E2 21542.543} C_VEL
LIN {X 0,Y 452.353,Z 732.377,A -85,B 0,C 180,E1 21540.85,E2 21540.85} C_VEL
LIN {X 0,Y 450.122,Z 750.175,A -85,B 0,C 180,E1 21539.035,E2 21539.035} C_VEL
LIN {X 0,Y 448.035,Z 766.456,A -85,B 0,C 180,E1 21537.073,E2 21537.073} C_VEL
LIN {X 0,Y 446.073,Z 781.749,A -85,B 0,C 180,E1 21534.922,E2 21534.922} C_VEL
LIN {X 0,Y 444.366,Z 795.798,A -85,B 0,C 180,E1 21532.628,E2 21532.628} C_VEL
LIN {X 0,Y 442.938,Z 808.364,A -85,B 0,C 180,E1 21530.204,E2 21530.204} C_VEL
LIN {X 0,Y 441.801,Z 819.563,A -85,B 0,C 180,E1 21527.653,E2 21527.653} C_VEL
LIN {X 0,Y 441.037,Z 828.427,A -85,B 0,C 180,E1 21525.246,E2 21525.246} C_VEL
LIN {X 0,Y 440.448,Z 836.292,A -85,B 0,C 180,E1 21522.542,E2 21522.542} C_VEL
LIN {X 0,Y 440.11,Z 843.027,A -85,B 0,C 180,E1 21519.608,E2 21519.608} C_VEL
LIN {X 0,Y 439.971,Z 847.638,A -85,B 0,C 180,E1 21516.918,E2 21516.918} C_VEL
LIN {X 0,Y 439.915,Z 850.672,A -85,B 0,C 180,E1 21514.171,E2 21514.171} C_VEL
LIN {X 0,Y 439.902,Z 852.257,A -85,B 0,C 180,E1 21511.433,E2 21511.433} C_VEL
LIN {X 0,Y 439.909,Z 852.302,A -85,B 0,C 180,E1 21508.828,E2 21508.828} C_VEL
LIN {X 0,Y 439.912,Z 850.782,A -85,B 0,C 180,E1 21505.96,E2 21505.96} C_VEL
LIN {X 0,Y 439.962,Z 847.817,A -85,B 0,C 180,E1 21503.213,E2 21503.213} C_VEL
LIN {X 0,Y 440.107,Z 843.145,A -85,B 0,C 180,E1 21500.454,E2 21500.454} C_VEL
LIN {X 0,Y 440.434,Z 836.527,A -85,B 0,C 180,E1 21497.546,E2 21497.546} C_VEL
LIN {X 0,Y 441.001,Z 828.853,A -85,B 0,C 180,E1 21494.887,E2 21494.887} C_VEL
LIN {X 0,Y 441.749,Z 820.098,A -85,B 0,C 180,E1 21492.481,E2 21492.481} C_VEL
LIN {X 0,Y 442.881,Z 808.941,A -85,B 0,C 180,E1 21489.912,E2 21489.912} C_VEL
LIN {X 0,Y 444.277,Z 796.533,A -85,B 0,C 180,E1 21487.506,E2 21487.506} C_VEL
LIN {X 0,Y 445.965,Z 782.641,A -85,B 0,C 180,E1 21485.213,E2 21485.213} C_VEL
LIN {X 0,Y 447.981,Z 766.882,A -85,B 0,C 180,E1 21482.98,E2 21482.98} C_VEL
LIN {X 0,Y 450.044,Z 750.763,A -85,B 0,C 180,E1 21481.032,E2 21481.032} C_VEL
LIN {X 0,Y 452.268,Z 733.092,A -85,B 0,C 180,E1 21479.218,E2 21479.218} C_VEL
LIN {X 0,Y 454.695,Z 712.859,A -85,B 0,C 180,E1 21477.456,E2 21477.456} C_VEL
LIN {X 0,Y 456.93,Z 693.277,A -85,B 0,C 180,E1 21476.03,E2 21476.03} C_VEL
LIN {X 0,Y 458.953,Z 673.058,A -85,B 0,C 180,E1 21474.815,E2 21474.815} C_VEL
LIN {X 0,Y 460.786,Z 652.597,A -85,B 0,C 180,E1 21473.823,E2 21473.823} C_VEL
LIN {X 0,Y 462.446,Z 630.802,A -85,B 0,C 180,E1 21472.992,E2 21472.992} C_VEL
LIN {X 0,Y 463.707,Z 609.374,A -85,B 0,C 180,E1 21472.396,E2 21472.396} C_VEL
LIN {X 0,Y 464.824,Z 571.672,A -85,B 0,C 180,E1 21471.699,E2 21471.699} C_VEL
LIN {X 0,Y 470.466,Z 355.176,A -85,B 0,C 180,E1 21467.91,E2 21467.91} C_VEL
LIN {X 0,Y 470.904,Z 331.781,A -85,B 0,C 180,E1 21467.483,E2 21467.483} C_VEL
LIN {X 0,Y 470.086,Z 327.758,A -85,B 0,C 180,E1 21467.318,E2 21467.318} C_VEL
LIN {X 0,Y 457.794,Z 307.448,A -85,B 0,C 180,E1 21465.577,E2 21465.577} C_VEL
LIN {X 0,Y 456.125,Z 304.406,A -85,B 0,C 180,E1 21465.253,E2 21465.253} C_VEL
LIN {X 0,Y 448.735,Z 288.673,A -85,B 0,C 180,E1 21462.811,E2 21462.811} C_VEL
LIN {X 0,Y 442.7,Z 276.525,A -85,B 0,C 180,E1 21460.747,E2 21460.747} C_VEL
LIN {X 0,Y 441.189,Z 273.014,A -85,B 0,C 180,E1 21460.089,E2 21460.089} C_VEL
LIN {X 0,Y 441.177,Z 272.739,A -85,B 0,C 180,E1 21456.653,E2 21456.653} C_VEL
LIN {X 0,Y 441.19,Z 272.755,A -85,B 0,C 180,E1 21452.95,E2 21452.95} C_VEL
LIN {X 0,Y 441.168,Z 272.769,A -85,B 0,C 180,E1 21449.245,E2 21449.245} C_VEL
LIN {X 0,Y 441.14,Z 272.781,A -85,B 0,C 180,E1 21445.571,E2 21445.571} C_VEL
LIN {X 0,Y 441.131,Z 272.783,A -85,B 0,C 180,E1 21441.821,E2 21441.821} C_VEL
LIN {X 0,Y 441.131,Z 272.784,A -85,B 0,C 180,E1 21438.09,E2 21438.09} C_VEL
LIN {X 0,Y 441.151,Z 272.777,A -85,B 0,C 180,E1 21434.437,E2 21434.437} C_VEL
LIN {X 0,Y 441.171,Z 272.77,A -85,B 0,C 180,E1 21430.71,E2 21430.71} C_VEL
LIN {X 0,Y 441.153,Z 272.769,A -85,B 0,C 180,E1 21427.03,E2 21427.03} C_VEL
LIN {X 0,Y 441.136,Z 272.773,A -85,B 0,C 180,E1 21423.378,E2 21423.378} C_VEL
LIN {X 0,Y 441.136,Z 272.781,A -85,B 0,C 180,E1 21419.61,E2 21419.61} C_VEL
LIN {X 0,Y 441.147,Z 272.781,A -85,B 0,C 180,E1 21415.841,E2 21415.841} C_VEL
LIN {X 0,Y 441.176,Z 272.78,A -85,B 0,C 180,E1 21412.184,E2 21412.184} C_VEL
LIN {X 0,Y 441.194,Z 272.772,A -85,B 0,C 180,E1 21408.496,E2 21408.496} C_VEL
LIN {X 0,Y 441.191,Z 272.767,A -85,B 0,C 180,E1 21404.758,E2 21404.758} C_VEL
LIN {X 0,Y 441.17,Z 272.767,A -85,B 0,C 180,E1 21401.089,E2 21401.089} C_VEL
LIN {X 0,Y 441.165,Z 272.768,A -85,B 0,C 180,E1 21397.338,E2 21397.338} C_VEL
LIN {X 0,Y 441.17,Z 272.768,A -85,B 0,C 180,E1 21393.533,E2 21393.533} C_VEL
LIN {X 0,Y 441.193,Z 272.742,A -85,B 0,C 180,E1 21389.944,E2 21389.944} C_VEL
LIN {X 0,Y 441.197,Z 272.776,A -85,B 0,C 180,E1 21386.117,E2 21386.117} C_VEL
LIN {X 0,Y 441.19,Z 272.737,A -85,B 0,C 180,E1 21382.27,E2 21382.27} C_VEL
LIN {X 0,Y 441.195,Z 272.745,A -85,B 0,C 180,E1 21378.567,E2 21378.567} C_VEL
LIN {X 0,Y 441.231,Z 273.04,A -85,B 0,C 180,E1 21376.759,E2 21376.759} C_VEL
LIN {X 0,Y 442.655,Z 276.488,A -85,B 0,C 180,E1 21376.096,E2 21376.096} C_VEL
LIN {X 0,Y 448.96,Z 289.785,A -85,B 0,C 180,E1 21373.724,E2 21373.724} C_VEL
LIN {X 0,Y 456.546,Z 307.38,A -85,B 0,C 180,E1 21370.905,E2 21370.905} C_VEL
LIN {X 0,Y 462.327,Z 322.096,A -85,B 0,C 180,E1 21368.769,E2 21368.769} C_VEL
LIN {X 0,Y 462.136,Z 326.767,A -85,B 0,C 180,E1 21368.405,E2 21368.405} C_VEL
LIN {X 0,Y 467.473,Z 358.737,A -85,B 0,C 180,E1 21367.235,E2 21367.235} C_VEL
LIN {X 0,Y 464.109,Z 529.829,A -85,B 0,C 180,E1 21364.469,E2 21364.469} C_VEL
LIN {X 0,Y 463.161,Z 537.528,A -85,B 0,C 180,E1 21364.422,E2 21364.422} C_VEL
LIN {X 0,Y 457.788,Z 558.055,A -85,B 0,C 180,E1 21364.562,E2 21364.562} C_VEL
LIN {X 0,Y 457.058,Z 564.663,A -85,B 0,C 180,E1 21364.513,E2 21364.513} C_VEL
LIN {X 0,Y 456.245,Z 596.589,A -85,B 0,C 180,E1 21363.95,E2 21363.95} C_VEL
LIN {X 0,Y 455.127,Z 616.834,A -85,B 0,C 180,E1 21363.383,E2 21363.383} C_VEL
LIN {X 0,Y 453.511,Z 636.806,A -85,B 0,C 180,E1 21362.584,E2 21362.584} C_VEL
LIN {X 0,Y 451.599,Z 655.845,A -85,B 0,C 180,E1 21361.585,E2 21361.585} C_VEL
LIN {X 0,Y 449.328,Z 674.768,A -85,B 0,C 180,E1 21360.339,E2 21360.339} C_VEL
LIN {X 0,Y 447.031,Z 691.864,A -85,B 0,C 180,E1 21358.962,E2 21358.962} C_VEL
LIN {X 0,Y 444.519,Z 708.837,A -85,B 0,C 180,E1 21357.313,E2 21357.313} C_VEL
LIN {X 0,Y 442.015,Z 724.715,A -85,B 0,C 180,E1 21355.453,E2 21355.453} C_VEL
LIN {X 0,Y 439.697,Z 739.096,A -85,B 0,C 180,E1 21353.449,E2 21353.449} C_VEL
LIN {X 0,Y 437.516,Z 752.852,A -85,B 0,C 180,E1 21351.166,E2 21351.166} C_VEL
LIN {X 0,Y 435.697,Z 765.02,A -85,B 0,C 180,E1 21348.74,E2 21348.74} C_VEL
LIN {X 0,Y 434.294,Z 775.37,A -85,B 0,C 180,E1 21346.251,E2 21346.251} C_VEL
LIN {X 0,Y 433.259,Z 784.334,A -85,B 0,C 180,E1 21343.614,E2 21343.614} C_VEL
LIN {X 0,Y 432.561,Z 791.915,A -85,B 0,C 180,E1 21340.791,E2 21340.791} C_VEL
LIN {X 0,Y 432.199,Z 797.469,A -85,B 0,C 180,E1 21338.049,E2 21338.049} C_VEL
LIN {X 0,Y 432.023,Z 801.365,A -85,B 0,C 180,E1 21335.312,E2 21335.312} C_VEL
LIN {X 0,Y 431.969,Z 803.704,A -85,B 0,C 180,E1 21332.521,E2 21332.521} C_VEL
LIN {X 0,Y 431.965,Z 804.441,A -85,B 0,C 180,E1 21329.867,E2 21329.867} C_VEL
LIN {X 0,Y 431.97,Z 803.556,A -85,B 0,C 180,E1 21327.081,E2 21327.081} C_VEL
LIN {X 0,Y 432.027,Z 801.164,A -85,B 0,C 180,E1 21324.422,E2 21324.422} C_VEL
LIN {X 0,Y 432.221,Z 797.028,A -85,B 0,C 180,E1 21321.62,E2 21321.62} C_VEL
LIN {X 0,Y 432.594,Z 791.465,A -85,B 0,C 180,E1 21318.94,E2 21318.94} C_VEL
LIN {X 0,Y 433.27,Z 784.197,A -85,B 0,C 180,E1 21316.25,E2 21316.25} C_VEL
LIN {X 0,Y 434.348,Z 774.988,A -85,B 0,C 180,E1 21313.553,E2 21313.553} C_VEL
LIN {X 0,Y 435.731,Z 764.809,A -85,B 0,C 180,E1 21311.123,E2 21311.123} C_VEL
LIN {X 0,Y 437.444,Z 753.33,A -85,B 0,C 180,E1 21308.831,E2 21308.831} C_VEL
LIN {X 0,Y 439.614,Z 739.667,A -85,B 0,C 180,E1 21306.546,E2 21306.546} C_VEL
LIN {X 0,Y 441.945,Z 725.199,A -85,B 0,C 180,E1 21304.516,E2 21304.516} C_VEL
LIN {X 0,Y 444.401,Z 709.619,A -85,B 0,C 180,E1 21302.68,E2 21302.68} C_VEL
LIN {X 0,Y 446.923,Z 692.611,A -85,B 0,C 180,E1 21301.015,E2 21301.015} C_VEL
LIN {X 0,Y 449.309,Z 674.982,A -85,B 0,C 180,E1 21299.586,E2 21299.586} C_VEL
LIN {X 0,Y 451.561,Z 656.272,A -85,B 0,C 180,E1 21298.348,E2 21298.348} C_VEL
LIN {X 0,Y 453.469,Z 637.444,A -85,B 0,C 180,E1 21297.353,E2 21297.353} C_VEL
LIN {X 0,Y 455.132,Z 616.904,A -85,B 0,C 180,E1 21296.528,E2 21296.528} C_VEL
LIN {X 0,Y 456.251,Z 596.693,A -85,B 0,C 180,E1 21295.96,E2 21295.96} C_VEL
LIN {X 0,Y 457.062,Z 565.187,A -85,B 0,C 180,E1 21295.403,E2 21295.403} C_VEL
LIN {X 0,Y 461.295,Z 359.102,A -85,B 0,C 180,E1 21292.033,E2 21292.033} C_VEL
LIN {X 0,Y 455.57,Z 325.423,A -85,B 0,C 180,E1 21290.733,E2 21290.733} C_VEL
LIN {X 0,Y 448.239,Z 306.982,A -85,B 0,C 180,E1 21287.971,E2 21287.971} C_VEL
LIN {X 0,Y 440.874,Z 290.172,A -85,B 0,C 180,E1 21285.146,E2 21285.146} C_VEL
LIN {X 0,Y 434.987,Z 277.818,A -85,B 0,C 180,E1 21282.842,E2 21282.842} C_VEL
LIN {X 0,Y 433.317,Z 274.16,A -85,B 0,C 180,E1 21282.111,E2 21282.111} C_VEL
LIN {X 0,Y 433.255,Z 273.733,A -85,B 0,C 180,E1 21281.302,E2 21281.302} C_VEL
LIN {X 0,Y 433.25,Z 273.723,A -85,B 0,C 180,E1 21277.536,E2 21277.536} C_VEL
LIN {X 0,Y 433.258,Z 273.764,A -85,B 0,C 180,E1 21273.792,E2 21273.792} C_VEL
LIN {X 0,Y 433.26,Z 273.73,A -85,B 0,C 180,E1 21269.899,E2 21269.899} C_VEL
LIN {X 0,Y 433.245,Z 273.755,A -85,B 0,C 180,E1 21266.14,E2 21266.14} C_VEL
LIN {X 0,Y 433.23,Z 273.756,A -85,B 0,C 180,E1 21262.384,E2 21262.384} C_VEL
LIN {X 0,Y 433.225,Z 273.756,A -85,B 0,C 180,E1 21258.572,E2 21258.572} C_VEL
LIN {X 0,Y 433.224,Z 273.755,A -85,B 0,C 180,E1 21254.76,E2 21254.76} C_VEL
LIN {X 0,Y 433.237,Z 273.756,A -85,B 0,C 180,E1 21251.044,E2 21251.044} C_VEL
LIN {X 0,Y 433.257,Z 273.762,A -85,B 0,C 180,E1 21247.292,E2 21247.292} C_VEL
LIN {X 0,Y 433.252,Z 273.77,A -85,B 0,C 180,E1 21243.44,E2 21243.44} C_VEL
LIN {X 0,Y 433.239,Z 273.768,A -85,B 0,C 180,E1 21239.604,E2 21239.604} C_VEL
LIN {X 0,Y 433.209,Z 273.766,A -85,B 0,C 180,E1 21235.897,E2 21235.897} C_VEL
LIN {X 0,Y 433.19,Z 273.761,A -85,B 0,C 180,E1 21232.307,E2 21232.307} C_VEL
LIN {X 0,Y 433.189,Z 273.758,A -85,B 0,C 180,E1 21228.551,E2 21228.551} C_VEL
LIN {X 0,Y 433.207,Z 273.757,A -85,B 0,C 180,E1 21224.882,E2 21224.882} C_VEL
LIN {X 0,Y 433.231,Z 273.757,A -85,B 0,C 180,E1 21221.123,E2 21221.123} C_VEL
LIN {X 0,Y 433.236,Z 273.758,A -85,B 0,C 180,E1 21217.331,E2 21217.331} C_VEL
LIN {X 0,Y 433.218,Z 273.761,A -85,B 0,C 180,E1 21213.549,E2 21213.549} C_VEL
LIN {X 0,Y 433.198,Z 273.738,A -85,B 0,C 180,E1 21209.941,E2 21209.941} C_VEL
LIN {X 0,Y 433.208,Z 273.774,A -85,B 0,C 180,E1 21206.188,E2 21206.188} C_VEL
LIN {X 0,Y 433.218,Z 273.732,A -85,B 0,C 180,E1 21202.461,E2 21202.461} C_VEL
LIN {X 0,Y 433.312,Z 274.092,A -85,B 0,C 180,E1 21200.955,E2 21200.955} C_VEL
LIN {X 0,Y 434.883,Z 277.743,A -85,B 0,C 180,E1 21200.271,E2 21200.271} C_VEL
LIN {X 0,Y 440.061,Z 287.909,A -85,B 0,C 180,E1 21198.437,E2 21198.437} C_VEL
LIN {X 0,Y 447.7,Z 304.051,A -85,B 0,C 180,E1 21195.797,E2 21195.797} C_VEL
LIN {X 0,Y 449.26,Z 306.968,A -85,B 0,C 180,E1 21195.422,E2 21195.422} C_VEL
LIN {X 0,Y 461.682,Z 327.22,A -85,B 0,C 180,E1 21193.58,E2 21193.58} C_VEL
LIN {X 0,Y 464.66,Z 332.666,A -85,B 0,C 180,E1 21193.148,E2 21193.148} C_VEL
LIN {X 0,Y 464.809,Z 337.438,A -85,B 0,C 180,E1 21193.033,E2 21193.033} C_VEL
LIN {X 0,Y 458.861,Z 550.687,A -85,B 0,C 180,E1 21189.25,E2 21189.25} C_VEL
LIN {X 0,Y 457.194,Z 607.721,A -85,B 0,C 180,E1 21188.21,E2 21188.21} C_VEL
LIN {X 0,Y 455.823,Z 629.655,A -85,B 0,C 180,E1 21187.598,E2 21187.598} C_VEL
LIN {X 0,Y 454.126,Z 650.861,A -85,B 0,C 180,E1 21186.788,E2 21186.788} C_VEL
LIN {X 0,Y 452.175,Z 671.333,A -85,B 0,C 180,E1 21185.792,E2 21185.792} C_VEL
LIN {X 0,Y 449.922,Z 692.259,A -85,B 0,C 180,E1 21184.518,E2 21184.518} C_VEL
LIN {X 0,Y 447.613,Z 711.508,A -85,B 0,C 180,E1 21183.107,E2 21183.107} C_VEL
LIN {X 0,Y 445.24,Z 730.343,A -85,B 0,C 180,E1 21181.473,E2 21181.473} C_VEL
LIN {X 0,Y 442.879,Z 748.359,A -85,B 0,C 180,E1 21179.631,E2 21179.631} C_VEL
LIN {X 0,Y 440.646,Z 764.761,A -85,B 0,C 180,E1 21177.651,E2 21177.651} C_VEL
LIN {X 0,Y 438.487,Z 780.885,A -85,B 0,C 180,E1 21175.383,E2 21175.383} C_VEL
LIN {X 0,Y 436.773,Z 794.277,A -85,B 0,C 180,E1 21173.187,E2 21173.187} C_VEL
LIN {X 0,Y 435.219,Z 806.997,A -85,B 0,C 180,E1 21170.719,E2 21170.719} C_VEL
LIN {X 0,Y 433.934,Z 818.922,A -85,B 0,C 180,E1 21167.984,E2 21167.984} C_VEL
LIN {X 0,Y 433.077,Z 828.386,A -85,B 0,C 180,E1 21165.396,E2 21165.396} C_VEL
LIN {X 0,Y 432.478,Z 836.405,A -85,B 0,C 180,E1 21162.675,E2 21162.675} C_VEL
LIN {X 0,Y 432.141,Z 842.638,A -85,B 0,C 180,E1 21159.993,E2 21159.993} C_VEL
LIN {X 0,Y 431.986,Z 847.225,A -85,B 0,C 180,E1 21157.313,E2 21157.313} C_VEL
LIN {X 0,Y 431.921,Z 850.444,A -85,B 0,C 180,E1 21154.514,E2 21154.514} C_VEL
LIN {X 0,Y 431.899,Z 852.209,A -85,B 0,C 180,E1 21151.725,E2 21151.725} C_VEL
LIN {X 0,Y 431.909,Z 852.347,A -85,B 0,C 180,E1 21149.072,E2 21149.072} C_VEL
LIN {X 0,Y 431.909,Z 851.122,A -85,B 0,C 180,E1 21146.284,E2 21146.284} C_VEL
LIN {X 0,Y 431.947,Z 848.455,A -85,B 0,C 180,E1 21143.621,E2 21143.621} C_VEL
LIN {X 0,Y 432.094,Z 843.907,A -85,B 0,C 180,E1 21140.678,E2 21140.678} C_VEL
